   // UNICODE_TO_GBK[19826] := 16#71EC;
   // UNICODE_TO_GBK[19827] := 16#A053;
   // UNICODE_TO_GBK[19828] := 16#71ED;
   // UNICODE_TO_GBK[19829] := 16#A054;
   // UNICODE_TO_GBK[19830] := 16#71EE;
   // UNICODE_TO_GBK[19831] := 16#DBC6;
   // UNICODE_TO_GBK[19832] := 16#71EF;
   // UNICODE_TO_GBK[19833] := 16#A055;
   // UNICODE_TO_GBK[19834] := 16#71F0;
   // UNICODE_TO_GBK[19835] := 16#A056;
   // UNICODE_TO_GBK[19836] := 16#71F1;
   // UNICODE_TO_GBK[19837] := 16#A057;
   // UNICODE_TO_GBK[19838] := 16#71F2;
   // UNICODE_TO_GBK[19839] := 16#A058;
   // UNICODE_TO_GBK[19840] := 16#71F3;
   // UNICODE_TO_GBK[19841] := 16#A059;
   // UNICODE_TO_GBK[19842] := 16#71F4;
   // UNICODE_TO_GBK[19843] := 16#A05A;
   // UNICODE_TO_GBK[19844] := 16#71F5;
   // UNICODE_TO_GBK[19845] := 16#A05B;
   // UNICODE_TO_GBK[19846] := 16#71F6;
   // UNICODE_TO_GBK[19847] := 16#A05C;
   // UNICODE_TO_GBK[19848] := 16#71F7;
   // UNICODE_TO_GBK[19849] := 16#A05D;
   // UNICODE_TO_GBK[19850] := 16#71F8;
   // UNICODE_TO_GBK[19851] := 16#A05E;
   // UNICODE_TO_GBK[19852] := 16#71F9;
   // UNICODE_TO_GBK[19853] := 16#ECDE;
   // UNICODE_TO_GBK[19854] := 16#71FA;
   // UNICODE_TO_GBK[19855] := 16#A05F;
   // UNICODE_TO_GBK[19856] := 16#71FB;
   // UNICODE_TO_GBK[19857] := 16#A060;
   // UNICODE_TO_GBK[19858] := 16#71FC;
   // UNICODE_TO_GBK[19859] := 16#A061;
   // UNICODE_TO_GBK[19860] := 16#71FD;
   // UNICODE_TO_GBK[19861] := 16#A062;
   // UNICODE_TO_GBK[19862] := 16#71FE;
   // UNICODE_TO_GBK[19863] := 16#A063;
   // UNICODE_TO_GBK[19864] := 16#71FF;
   // UNICODE_TO_GBK[19865] := 16#A064;
   // UNICODE_TO_GBK[19866] := 16#7200;
   // UNICODE_TO_GBK[19867] := 16#A065;
   // UNICODE_TO_GBK[19868] := 16#7201;
   // UNICODE_TO_GBK[19869] := 16#A066;
   // UNICODE_TO_GBK[19870] := 16#7202;
   // UNICODE_TO_GBK[19871] := 16#A067;
   // UNICODE_TO_GBK[19872] := 16#7203;
   // UNICODE_TO_GBK[19873] := 16#A068;
   // UNICODE_TO_GBK[19874] := 16#7204;
   // UNICODE_TO_GBK[19875] := 16#A069;
   // UNICODE_TO_GBK[19876] := 16#7205;
   // UNICODE_TO_GBK[19877] := 16#A06A;
   // UNICODE_TO_GBK[19878] := 16#7206;
   // UNICODE_TO_GBK[19879] := 16#B1AC;
   // UNICODE_TO_GBK[19880] := 16#7207;
   // UNICODE_TO_GBK[19881] := 16#A06B;
   // UNICODE_TO_GBK[19882] := 16#7208;
   // UNICODE_TO_GBK[19883] := 16#A06C;
   // UNICODE_TO_GBK[19884] := 16#7209;
   // UNICODE_TO_GBK[19885] := 16#A06D;
   // UNICODE_TO_GBK[19886] := 16#720A;
   // UNICODE_TO_GBK[19887] := 16#A06E;
   // UNICODE_TO_GBK[19888] := 16#720B;
   // UNICODE_TO_GBK[19889] := 16#A06F;
   // UNICODE_TO_GBK[19890] := 16#720C;
   // UNICODE_TO_GBK[19891] := 16#A070;
   // UNICODE_TO_GBK[19892] := 16#720D;
   // UNICODE_TO_GBK[19893] := 16#A071;
   // UNICODE_TO_GBK[19894] := 16#720E;
   // UNICODE_TO_GBK[19895] := 16#A072;
   // UNICODE_TO_GBK[19896] := 16#720F;
   // UNICODE_TO_GBK[19897] := 16#A073;
   // UNICODE_TO_GBK[19898] := 16#7210;
   // UNICODE_TO_GBK[19899] := 16#A074;
   // UNICODE_TO_GBK[19900] := 16#7211;
   // UNICODE_TO_GBK[19901] := 16#A075;
   // UNICODE_TO_GBK[19902] := 16#7212;
   // UNICODE_TO_GBK[19903] := 16#A076;
   // UNICODE_TO_GBK[19904] := 16#7213;
   // UNICODE_TO_GBK[19905] := 16#A077;
   // UNICODE_TO_GBK[19906] := 16#7214;
   // UNICODE_TO_GBK[19907] := 16#A078;
   // UNICODE_TO_GBK[19908] := 16#7215;
   // UNICODE_TO_GBK[19909] := 16#A079;
   // UNICODE_TO_GBK[19910] := 16#7216;
   // UNICODE_TO_GBK[19911] := 16#A07A;
   // UNICODE_TO_GBK[19912] := 16#7217;
   // UNICODE_TO_GBK[19913] := 16#A07B;
   // UNICODE_TO_GBK[19914] := 16#7218;
   // UNICODE_TO_GBK[19915] := 16#A07C;
   // UNICODE_TO_GBK[19916] := 16#7219;
   // UNICODE_TO_GBK[19917] := 16#A07D;
   // UNICODE_TO_GBK[19918] := 16#721A;
   // UNICODE_TO_GBK[19919] := 16#A07E;
   // UNICODE_TO_GBK[19920] := 16#721B;
   // UNICODE_TO_GBK[19921] := 16#A080;
   // UNICODE_TO_GBK[19922] := 16#721C;
   // UNICODE_TO_GBK[19923] := 16#A081;
   // UNICODE_TO_GBK[19924] := 16#721D;
   // UNICODE_TO_GBK[19925] := 16#ECDF;
   // UNICODE_TO_GBK[19926] := 16#721E;
   // UNICODE_TO_GBK[19927] := 16#A082;
   // UNICODE_TO_GBK[19928] := 16#721F;
   // UNICODE_TO_GBK[19929] := 16#A083;
   // UNICODE_TO_GBK[19930] := 16#7220;
   // UNICODE_TO_GBK[19931] := 16#A084;
   // UNICODE_TO_GBK[19932] := 16#7221;
   // UNICODE_TO_GBK[19933] := 16#A085;
   // UNICODE_TO_GBK[19934] := 16#7222;
   // UNICODE_TO_GBK[19935] := 16#A086;
   // UNICODE_TO_GBK[19936] := 16#7223;
   // UNICODE_TO_GBK[19937] := 16#A087;
   // UNICODE_TO_GBK[19938] := 16#7224;
   // UNICODE_TO_GBK[19939] := 16#A088;
   // UNICODE_TO_GBK[19940] := 16#7225;
   // UNICODE_TO_GBK[19941] := 16#A089;
   // UNICODE_TO_GBK[19942] := 16#7226;
   // UNICODE_TO_GBK[19943] := 16#A08A;
   // UNICODE_TO_GBK[19944] := 16#7227;
   // UNICODE_TO_GBK[19945] := 16#A08B;
   // UNICODE_TO_GBK[19946] := 16#7228;
   // UNICODE_TO_GBK[19947] := 16#ECE0;
   // UNICODE_TO_GBK[19948] := 16#7229;
   // UNICODE_TO_GBK[19949] := 16#A08C;
   // UNICODE_TO_GBK[19950] := 16#722A;
   // UNICODE_TO_GBK[19951] := 16#D7A6;
   // UNICODE_TO_GBK[19952] := 16#722B;
   // UNICODE_TO_GBK[19953] := 16#A08D;
   // UNICODE_TO_GBK[19954] := 16#722C;
   // UNICODE_TO_GBK[19955] := 16#C5C0;
   // UNICODE_TO_GBK[19956] := 16#722D;
   // UNICODE_TO_GBK[19957] := 16#A08E;
   // UNICODE_TO_GBK[19958] := 16#722E;
   // UNICODE_TO_GBK[19959] := 16#A08F;
   // UNICODE_TO_GBK[19960] := 16#722F;
   // UNICODE_TO_GBK[19961] := 16#A090;
   // UNICODE_TO_GBK[19962] := 16#7230;
   // UNICODE_TO_GBK[19963] := 16#EBBC;
   // UNICODE_TO_GBK[19964] := 16#7231;
   // UNICODE_TO_GBK[19965] := 16#B0AE;
   // UNICODE_TO_GBK[19966] := 16#7232;
   // UNICODE_TO_GBK[19967] := 16#A091;
   // UNICODE_TO_GBK[19968] := 16#7233;
   // UNICODE_TO_GBK[19969] := 16#A092;
   // UNICODE_TO_GBK[19970] := 16#7234;
   // UNICODE_TO_GBK[19971] := 16#A093;
   // UNICODE_TO_GBK[19972] := 16#7235;
   // UNICODE_TO_GBK[19973] := 16#BEF4;
   // UNICODE_TO_GBK[19974] := 16#7236;
   // UNICODE_TO_GBK[19975] := 16#B8B8;
   // UNICODE_TO_GBK[19976] := 16#7237;
   // UNICODE_TO_GBK[19977] := 16#D2AF;
   // UNICODE_TO_GBK[19978] := 16#7238;
   // UNICODE_TO_GBK[19979] := 16#B0D6;
   // UNICODE_TO_GBK[19980] := 16#7239;
   // UNICODE_TO_GBK[19981] := 16#B5F9;
   // UNICODE_TO_GBK[19982] := 16#723A;
   // UNICODE_TO_GBK[19983] := 16#A094;
   // UNICODE_TO_GBK[19984] := 16#723B;
   // UNICODE_TO_GBK[19985] := 16#D8B3;
   // UNICODE_TO_GBK[19986] := 16#723C;
   // UNICODE_TO_GBK[19987] := 16#A095;
   // UNICODE_TO_GBK[19988] := 16#723D;
   // UNICODE_TO_GBK[19989] := 16#CBAC;
   // UNICODE_TO_GBK[19990] := 16#723E;
   // UNICODE_TO_GBK[19991] := 16#A096;
   // UNICODE_TO_GBK[19992] := 16#723F;
   // UNICODE_TO_GBK[19993] := 16#E3DD;
   // UNICODE_TO_GBK[19994] := 16#7240;
   // UNICODE_TO_GBK[19995] := 16#A097;
   // UNICODE_TO_GBK[19996] := 16#7241;
   // UNICODE_TO_GBK[19997] := 16#A098;
   // UNICODE_TO_GBK[19998] := 16#7242;
   // UNICODE_TO_GBK[19999] := 16#A099;
   // UNICODE_TO_GBK[20000] := 16#7243;
   // UNICODE_TO_GBK[20001] := 16#A09A;
   // UNICODE_TO_GBK[20002] := 16#7244;
   // UNICODE_TO_GBK[20003] := 16#A09B;
   // UNICODE_TO_GBK[20004] := 16#7245;
   // UNICODE_TO_GBK[20005] := 16#A09C;
   // UNICODE_TO_GBK[20006] := 16#7246;
   // UNICODE_TO_GBK[20007] := 16#A09D;
   // UNICODE_TO_GBK[20008] := 16#7247;
   // UNICODE_TO_GBK[20009] := 16#C6AC;
   // UNICODE_TO_GBK[20010] := 16#7248;
   // UNICODE_TO_GBK[20011] := 16#B0E6;
   // UNICODE_TO_GBK[20012] := 16#7249;
   // UNICODE_TO_GBK[20013] := 16#A09E;
   // UNICODE_TO_GBK[20014] := 16#724A;
   // UNICODE_TO_GBK[20015] := 16#A09F;
   // UNICODE_TO_GBK[20016] := 16#724B;
   // UNICODE_TO_GBK[20017] := 16#A0A0;
   // UNICODE_TO_GBK[20018] := 16#724C;
   // UNICODE_TO_GBK[20019] := 16#C5C6;
   // UNICODE_TO_GBK[20020] := 16#724D;
   // UNICODE_TO_GBK[20021] := 16#EBB9;
   // UNICODE_TO_GBK[20022] := 16#724E;
   // UNICODE_TO_GBK[20023] := 16#A0A1;
   // UNICODE_TO_GBK[20024] := 16#724F;
   // UNICODE_TO_GBK[20025] := 16#A0A2;
   // UNICODE_TO_GBK[20026] := 16#7250;
   // UNICODE_TO_GBK[20027] := 16#A0A3;
   // UNICODE_TO_GBK[20028] := 16#7251;
   // UNICODE_TO_GBK[20029] := 16#A0A4;
   // UNICODE_TO_GBK[20030] := 16#7252;
   // UNICODE_TO_GBK[20031] := 16#EBBA;
   // UNICODE_TO_GBK[20032] := 16#7253;
   // UNICODE_TO_GBK[20033] := 16#A0A5;
   // UNICODE_TO_GBK[20034] := 16#7254;
   // UNICODE_TO_GBK[20035] := 16#A0A6;
   // UNICODE_TO_GBK[20036] := 16#7255;
   // UNICODE_TO_GBK[20037] := 16#A0A7;
   // UNICODE_TO_GBK[20038] := 16#7256;
   // UNICODE_TO_GBK[20039] := 16#EBBB;
   // UNICODE_TO_GBK[20040] := 16#7257;
   // UNICODE_TO_GBK[20041] := 16#A0A8;
   // UNICODE_TO_GBK[20042] := 16#7258;
   // UNICODE_TO_GBK[20043] := 16#A0A9;
   // UNICODE_TO_GBK[20044] := 16#7259;
   // UNICODE_TO_GBK[20045] := 16#D1C0;
   // UNICODE_TO_GBK[20046] := 16#725A;
   // UNICODE_TO_GBK[20047] := 16#A0AA;
   // UNICODE_TO_GBK[20048] := 16#725B;
   // UNICODE_TO_GBK[20049] := 16#C5A3;
   // UNICODE_TO_GBK[20050] := 16#725C;
   // UNICODE_TO_GBK[20051] := 16#A0AB;
   // UNICODE_TO_GBK[20052] := 16#725D;
   // UNICODE_TO_GBK[20053] := 16#EAF2;
   // UNICODE_TO_GBK[20054] := 16#725E;
   // UNICODE_TO_GBK[20055] := 16#A0AC;
   // UNICODE_TO_GBK[20056] := 16#725F;
   // UNICODE_TO_GBK[20057] := 16#C4B2;
   // UNICODE_TO_GBK[20058] := 16#7260;
   // UNICODE_TO_GBK[20059] := 16#A0AD;
   // UNICODE_TO_GBK[20060] := 16#7261;
   // UNICODE_TO_GBK[20061] := 16#C4B5;
   // UNICODE_TO_GBK[20062] := 16#7262;
   // UNICODE_TO_GBK[20063] := 16#C0CE;
   // UNICODE_TO_GBK[20064] := 16#7263;
   // UNICODE_TO_GBK[20065] := 16#A0AE;
   // UNICODE_TO_GBK[20066] := 16#7264;
   // UNICODE_TO_GBK[20067] := 16#A0AF;
   // UNICODE_TO_GBK[20068] := 16#7265;
   // UNICODE_TO_GBK[20069] := 16#A0B0;
   // UNICODE_TO_GBK[20070] := 16#7266;
   // UNICODE_TO_GBK[20071] := 16#EAF3;
   // UNICODE_TO_GBK[20072] := 16#7267;
   // UNICODE_TO_GBK[20073] := 16#C4C1;
   // UNICODE_TO_GBK[20074] := 16#7268;
   // UNICODE_TO_GBK[20075] := 16#A0B1;
   // UNICODE_TO_GBK[20076] := 16#7269;
   // UNICODE_TO_GBK[20077] := 16#CEEF;
   // UNICODE_TO_GBK[20078] := 16#726A;
   // UNICODE_TO_GBK[20079] := 16#A0B2;
   // UNICODE_TO_GBK[20080] := 16#726B;
   // UNICODE_TO_GBK[20081] := 16#A0B3;
   // UNICODE_TO_GBK[20082] := 16#726C;
   // UNICODE_TO_GBK[20083] := 16#A0B4;
   // UNICODE_TO_GBK[20084] := 16#726D;
   // UNICODE_TO_GBK[20085] := 16#A0B5;
   // UNICODE_TO_GBK[20086] := 16#726E;
   // UNICODE_TO_GBK[20087] := 16#EAF0;
   // UNICODE_TO_GBK[20088] := 16#726F;
   // UNICODE_TO_GBK[20089] := 16#EAF4;
   // UNICODE_TO_GBK[20090] := 16#7270;
   // UNICODE_TO_GBK[20091] := 16#A0B6;
   // UNICODE_TO_GBK[20092] := 16#7271;
   // UNICODE_TO_GBK[20093] := 16#A0B7;
   // UNICODE_TO_GBK[20094] := 16#7272;
   // UNICODE_TO_GBK[20095] := 16#C9FC;
   // UNICODE_TO_GBK[20096] := 16#7273;
   // UNICODE_TO_GBK[20097] := 16#A0B8;
   // UNICODE_TO_GBK[20098] := 16#7274;
   // UNICODE_TO_GBK[20099] := 16#A0B9;
   // UNICODE_TO_GBK[20100] := 16#7275;
   // UNICODE_TO_GBK[20101] := 16#C7A3;
   // UNICODE_TO_GBK[20102] := 16#7276;
   // UNICODE_TO_GBK[20103] := 16#A0BA;
   // UNICODE_TO_GBK[20104] := 16#7277;
   // UNICODE_TO_GBK[20105] := 16#A0BB;
   // UNICODE_TO_GBK[20106] := 16#7278;
   // UNICODE_TO_GBK[20107] := 16#A0BC;
   // UNICODE_TO_GBK[20108] := 16#7279;
   // UNICODE_TO_GBK[20109] := 16#CCD8;
   // UNICODE_TO_GBK[20110] := 16#727A;
   // UNICODE_TO_GBK[20111] := 16#CEFE;
   // UNICODE_TO_GBK[20112] := 16#727B;
   // UNICODE_TO_GBK[20113] := 16#A0BD;
   // UNICODE_TO_GBK[20114] := 16#727C;
   // UNICODE_TO_GBK[20115] := 16#A0BE;
   // UNICODE_TO_GBK[20116] := 16#727D;
   // UNICODE_TO_GBK[20117] := 16#A0BF;
   // UNICODE_TO_GBK[20118] := 16#727E;
   // UNICODE_TO_GBK[20119] := 16#EAF5;
   // UNICODE_TO_GBK[20120] := 16#727F;
   // UNICODE_TO_GBK[20121] := 16#EAF6;
   // UNICODE_TO_GBK[20122] := 16#7280;
   // UNICODE_TO_GBK[20123] := 16#CFAC;
   // UNICODE_TO_GBK[20124] := 16#7281;
   // UNICODE_TO_GBK[20125] := 16#C0E7;
   // UNICODE_TO_GBK[20126] := 16#7282;
   // UNICODE_TO_GBK[20127] := 16#A0C0;
   // UNICODE_TO_GBK[20128] := 16#7283;
   // UNICODE_TO_GBK[20129] := 16#A0C1;
   // UNICODE_TO_GBK[20130] := 16#7284;
   // UNICODE_TO_GBK[20131] := 16#EAF7;
   // UNICODE_TO_GBK[20132] := 16#7285;
   // UNICODE_TO_GBK[20133] := 16#A0C2;
   // UNICODE_TO_GBK[20134] := 16#7286;
   // UNICODE_TO_GBK[20135] := 16#A0C3;
   // UNICODE_TO_GBK[20136] := 16#7287;
   // UNICODE_TO_GBK[20137] := 16#A0C4;
   // UNICODE_TO_GBK[20138] := 16#7288;
   // UNICODE_TO_GBK[20139] := 16#A0C5;
   // UNICODE_TO_GBK[20140] := 16#7289;
   // UNICODE_TO_GBK[20141] := 16#A0C6;
   // UNICODE_TO_GBK[20142] := 16#728A;
   // UNICODE_TO_GBK[20143] := 16#B6BF;
   // UNICODE_TO_GBK[20144] := 16#728B;
   // UNICODE_TO_GBK[20145] := 16#EAF8;
   // UNICODE_TO_GBK[20146] := 16#728C;
   // UNICODE_TO_GBK[20147] := 16#A0C7;
   // UNICODE_TO_GBK[20148] := 16#728D;
   // UNICODE_TO_GBK[20149] := 16#EAF9;
   // UNICODE_TO_GBK[20150] := 16#728E;
   // UNICODE_TO_GBK[20151] := 16#A0C8;
   // UNICODE_TO_GBK[20152] := 16#728F;
   // UNICODE_TO_GBK[20153] := 16#EAFA;
   // UNICODE_TO_GBK[20154] := 16#7290;
   // UNICODE_TO_GBK[20155] := 16#A0C9;
   // UNICODE_TO_GBK[20156] := 16#7291;
   // UNICODE_TO_GBK[20157] := 16#A0CA;
   // UNICODE_TO_GBK[20158] := 16#7292;
   // UNICODE_TO_GBK[20159] := 16#EAFB;
   // UNICODE_TO_GBK[20160] := 16#7293;
   // UNICODE_TO_GBK[20161] := 16#A0CB;
   // UNICODE_TO_GBK[20162] := 16#7294;
   // UNICODE_TO_GBK[20163] := 16#A0CC;
   // UNICODE_TO_GBK[20164] := 16#7295;
   // UNICODE_TO_GBK[20165] := 16#A0CD;
   // UNICODE_TO_GBK[20166] := 16#7296;
   // UNICODE_TO_GBK[20167] := 16#A0CE;
   // UNICODE_TO_GBK[20168] := 16#7297;
   // UNICODE_TO_GBK[20169] := 16#A0CF;
   // UNICODE_TO_GBK[20170] := 16#7298;
   // UNICODE_TO_GBK[20171] := 16#A0D0;
   // UNICODE_TO_GBK[20172] := 16#7299;
   // UNICODE_TO_GBK[20173] := 16#A0D1;
   // UNICODE_TO_GBK[20174] := 16#729A;
   // UNICODE_TO_GBK[20175] := 16#A0D2;
   // UNICODE_TO_GBK[20176] := 16#729B;
   // UNICODE_TO_GBK[20177] := 16#A0D3;
   // UNICODE_TO_GBK[20178] := 16#729C;
   // UNICODE_TO_GBK[20179] := 16#A0D4;
   // UNICODE_TO_GBK[20180] := 16#729D;
   // UNICODE_TO_GBK[20181] := 16#A0D5;
   // UNICODE_TO_GBK[20182] := 16#729E;
   // UNICODE_TO_GBK[20183] := 16#A0D6;
   // UNICODE_TO_GBK[20184] := 16#729F;
   // UNICODE_TO_GBK[20185] := 16#EAF1;
   // UNICODE_TO_GBK[20186] := 16#72A0;
   // UNICODE_TO_GBK[20187] := 16#A0D7;
   // UNICODE_TO_GBK[20188] := 16#72A1;
   // UNICODE_TO_GBK[20189] := 16#A0D8;
   // UNICODE_TO_GBK[20190] := 16#72A2;
   // UNICODE_TO_GBK[20191] := 16#A0D9;
   // UNICODE_TO_GBK[20192] := 16#72A3;
   // UNICODE_TO_GBK[20193] := 16#A0DA;
   // UNICODE_TO_GBK[20194] := 16#72A4;
   // UNICODE_TO_GBK[20195] := 16#A0DB;
   // UNICODE_TO_GBK[20196] := 16#72A5;
   // UNICODE_TO_GBK[20197] := 16#A0DC;
   // UNICODE_TO_GBK[20198] := 16#72A6;
   // UNICODE_TO_GBK[20199] := 16#A0DD;
   // UNICODE_TO_GBK[20200] := 16#72A7;
   // UNICODE_TO_GBK[20201] := 16#A0DE;
   // UNICODE_TO_GBK[20202] := 16#72A8;
   // UNICODE_TO_GBK[20203] := 16#A0DF;
   // UNICODE_TO_GBK[20204] := 16#72A9;
   // UNICODE_TO_GBK[20205] := 16#A0E0;
   // UNICODE_TO_GBK[20206] := 16#72AA;
   // UNICODE_TO_GBK[20207] := 16#A0E1;
   // UNICODE_TO_GBK[20208] := 16#72AB;
   // UNICODE_TO_GBK[20209] := 16#A0E2;
   // UNICODE_TO_GBK[20210] := 16#72AC;
   // UNICODE_TO_GBK[20211] := 16#C8AE;
   // UNICODE_TO_GBK[20212] := 16#72AD;
   // UNICODE_TO_GBK[20213] := 16#E1EB;
   // UNICODE_TO_GBK[20214] := 16#72AE;
   // UNICODE_TO_GBK[20215] := 16#A0E3;
   // UNICODE_TO_GBK[20216] := 16#72AF;
   // UNICODE_TO_GBK[20217] := 16#B7B8;
   // UNICODE_TO_GBK[20218] := 16#72B0;
   // UNICODE_TO_GBK[20219] := 16#E1EC;
   // UNICODE_TO_GBK[20220] := 16#72B1;
   // UNICODE_TO_GBK[20221] := 16#A0E4;
   // UNICODE_TO_GBK[20222] := 16#72B2;
   // UNICODE_TO_GBK[20223] := 16#A0E5;
   // UNICODE_TO_GBK[20224] := 16#72B3;
   // UNICODE_TO_GBK[20225] := 16#A0E6;
   // UNICODE_TO_GBK[20226] := 16#72B4;
   // UNICODE_TO_GBK[20227] := 16#E1ED;
   // UNICODE_TO_GBK[20228] := 16#72B5;
   // UNICODE_TO_GBK[20229] := 16#A0E7;
   // UNICODE_TO_GBK[20230] := 16#72B6;
   // UNICODE_TO_GBK[20231] := 16#D7B4;
   // UNICODE_TO_GBK[20232] := 16#72B7;
   // UNICODE_TO_GBK[20233] := 16#E1EE;
   // UNICODE_TO_GBK[20234] := 16#72B8;
   // UNICODE_TO_GBK[20235] := 16#E1EF;
   // UNICODE_TO_GBK[20236] := 16#72B9;
   // UNICODE_TO_GBK[20237] := 16#D3CC;
   // UNICODE_TO_GBK[20238] := 16#72BA;
   // UNICODE_TO_GBK[20239] := 16#A0E8;
   // UNICODE_TO_GBK[20240] := 16#72BB;
   // UNICODE_TO_GBK[20241] := 16#A0E9;
   // UNICODE_TO_GBK[20242] := 16#72BC;
   // UNICODE_TO_GBK[20243] := 16#A0EA;
   // UNICODE_TO_GBK[20244] := 16#72BD;
   // UNICODE_TO_GBK[20245] := 16#A0EB;
   // UNICODE_TO_GBK[20246] := 16#72BE;
   // UNICODE_TO_GBK[20247] := 16#A0EC;
   // UNICODE_TO_GBK[20248] := 16#72BF;
   // UNICODE_TO_GBK[20249] := 16#A0ED;
   // UNICODE_TO_GBK[20250] := 16#72C0;
   // UNICODE_TO_GBK[20251] := 16#A0EE;
   // UNICODE_TO_GBK[20252] := 16#72C1;
   // UNICODE_TO_GBK[20253] := 16#E1F1;
   // UNICODE_TO_GBK[20254] := 16#72C2;
   // UNICODE_TO_GBK[20255] := 16#BFF1;
   // UNICODE_TO_GBK[20256] := 16#72C3;
   // UNICODE_TO_GBK[20257] := 16#E1F0;
   // UNICODE_TO_GBK[20258] := 16#72C4;
   // UNICODE_TO_GBK[20259] := 16#B5D2;
   // UNICODE_TO_GBK[20260] := 16#72C5;
   // UNICODE_TO_GBK[20261] := 16#A0EF;
   // UNICODE_TO_GBK[20262] := 16#72C6;
   // UNICODE_TO_GBK[20263] := 16#A0F0;
   // UNICODE_TO_GBK[20264] := 16#72C7;
   // UNICODE_TO_GBK[20265] := 16#A0F1;
   // UNICODE_TO_GBK[20266] := 16#72C8;
   // UNICODE_TO_GBK[20267] := 16#B1B7;
   // UNICODE_TO_GBK[20268] := 16#72C9;
   // UNICODE_TO_GBK[20269] := 16#A0F2;
   // UNICODE_TO_GBK[20270] := 16#72CA;
   // UNICODE_TO_GBK[20271] := 16#A0F3;
   // UNICODE_TO_GBK[20272] := 16#72CB;
   // UNICODE_TO_GBK[20273] := 16#A0F4;
   // UNICODE_TO_GBK[20274] := 16#72CC;
   // UNICODE_TO_GBK[20275] := 16#A0F5;
   // UNICODE_TO_GBK[20276] := 16#72CD;
   // UNICODE_TO_GBK[20277] := 16#E1F3;
   // UNICODE_TO_GBK[20278] := 16#72CE;
   // UNICODE_TO_GBK[20279] := 16#E1F2;
   // UNICODE_TO_GBK[20280] := 16#72CF;
   // UNICODE_TO_GBK[20281] := 16#A0F6;
   // UNICODE_TO_GBK[20282] := 16#72D0;
   // UNICODE_TO_GBK[20283] := 16#BAFC;
   // UNICODE_TO_GBK[20284] := 16#72D1;
   // UNICODE_TO_GBK[20285] := 16#A0F7;
   // UNICODE_TO_GBK[20286] := 16#72D2;
   // UNICODE_TO_GBK[20287] := 16#E1F4;
   // UNICODE_TO_GBK[20288] := 16#72D3;
   // UNICODE_TO_GBK[20289] := 16#A0F8;
   // UNICODE_TO_GBK[20290] := 16#72D4;
   // UNICODE_TO_GBK[20291] := 16#A0F9;
   // UNICODE_TO_GBK[20292] := 16#72D5;
   // UNICODE_TO_GBK[20293] := 16#A0FA;
   // UNICODE_TO_GBK[20294] := 16#72D6;
   // UNICODE_TO_GBK[20295] := 16#A0FB;
   // UNICODE_TO_GBK[20296] := 16#72D7;
   // UNICODE_TO_GBK[20297] := 16#B9B7;
   // UNICODE_TO_GBK[20298] := 16#72D8;
   // UNICODE_TO_GBK[20299] := 16#A0FC;
   // UNICODE_TO_GBK[20300] := 16#72D9;
   // UNICODE_TO_GBK[20301] := 16#BED1;
   // UNICODE_TO_GBK[20302] := 16#72DA;
   // UNICODE_TO_GBK[20303] := 16#A0FD;
   // UNICODE_TO_GBK[20304] := 16#72DB;
   // UNICODE_TO_GBK[20305] := 16#A0FE;
   // UNICODE_TO_GBK[20306] := 16#72DC;
   // UNICODE_TO_GBK[20307] := 16#AA40;
   // UNICODE_TO_GBK[20308] := 16#72DD;
   // UNICODE_TO_GBK[20309] := 16#AA41;
   // UNICODE_TO_GBK[20310] := 16#72DE;
   // UNICODE_TO_GBK[20311] := 16#C4FC;
   // UNICODE_TO_GBK[20312] := 16#72DF;
   // UNICODE_TO_GBK[20313] := 16#AA42;
   // UNICODE_TO_GBK[20314] := 16#72E0;
   // UNICODE_TO_GBK[20315] := 16#BADD;
   // UNICODE_TO_GBK[20316] := 16#72E1;
   // UNICODE_TO_GBK[20317] := 16#BDC6;
   // UNICODE_TO_GBK[20318] := 16#72E2;
   // UNICODE_TO_GBK[20319] := 16#AA43;
   // UNICODE_TO_GBK[20320] := 16#72E3;
   // UNICODE_TO_GBK[20321] := 16#AA44;
   // UNICODE_TO_GBK[20322] := 16#72E4;
   // UNICODE_TO_GBK[20323] := 16#AA45;
   // UNICODE_TO_GBK[20324] := 16#72E5;
   // UNICODE_TO_GBK[20325] := 16#AA46;
   // UNICODE_TO_GBK[20326] := 16#72E6;
   // UNICODE_TO_GBK[20327] := 16#AA47;
   // UNICODE_TO_GBK[20328] := 16#72E7;
   // UNICODE_TO_GBK[20329] := 16#AA48;
   // UNICODE_TO_GBK[20330] := 16#72E8;
   // UNICODE_TO_GBK[20331] := 16#E1F5;
   // UNICODE_TO_GBK[20332] := 16#72E9;
   // UNICODE_TO_GBK[20333] := 16#E1F7;
   // UNICODE_TO_GBK[20334] := 16#72EA;
   // UNICODE_TO_GBK[20335] := 16#AA49;
   // UNICODE_TO_GBK[20336] := 16#72EB;
   // UNICODE_TO_GBK[20337] := 16#AA4A;
   // UNICODE_TO_GBK[20338] := 16#72EC;
   // UNICODE_TO_GBK[20339] := 16#B6C0;
   // UNICODE_TO_GBK[20340] := 16#72ED;
   // UNICODE_TO_GBK[20341] := 16#CFC1;
   // UNICODE_TO_GBK[20342] := 16#72EE;
   // UNICODE_TO_GBK[20343] := 16#CAA8;
   // UNICODE_TO_GBK[20344] := 16#72EF;
   // UNICODE_TO_GBK[20345] := 16#E1F6;
   // UNICODE_TO_GBK[20346] := 16#72F0;
   // UNICODE_TO_GBK[20347] := 16#D5F8;
   // UNICODE_TO_GBK[20348] := 16#72F1;
   // UNICODE_TO_GBK[20349] := 16#D3FC;
   // UNICODE_TO_GBK[20350] := 16#72F2;
   // UNICODE_TO_GBK[20351] := 16#E1F8;
   // UNICODE_TO_GBK[20352] := 16#72F3;
   // UNICODE_TO_GBK[20353] := 16#E1FC;
   // UNICODE_TO_GBK[20354] := 16#72F4;
   // UNICODE_TO_GBK[20355] := 16#E1F9;
   // UNICODE_TO_GBK[20356] := 16#72F5;
   // UNICODE_TO_GBK[20357] := 16#AA4B;
   // UNICODE_TO_GBK[20358] := 16#72F6;
   // UNICODE_TO_GBK[20359] := 16#AA4C;
   // UNICODE_TO_GBK[20360] := 16#72F7;
   // UNICODE_TO_GBK[20361] := 16#E1FA;
   // UNICODE_TO_GBK[20362] := 16#72F8;
   // UNICODE_TO_GBK[20363] := 16#C0EA;
   // UNICODE_TO_GBK[20364] := 16#72F9;
   // UNICODE_TO_GBK[20365] := 16#AA4D;
   // UNICODE_TO_GBK[20366] := 16#72FA;
   // UNICODE_TO_GBK[20367] := 16#E1FE;
   // UNICODE_TO_GBK[20368] := 16#72FB;
   // UNICODE_TO_GBK[20369] := 16#E2A1;
   // UNICODE_TO_GBK[20370] := 16#72FC;
   // UNICODE_TO_GBK[20371] := 16#C0C7;
   // UNICODE_TO_GBK[20372] := 16#72FD;
   // UNICODE_TO_GBK[20373] := 16#AA4E;
   // UNICODE_TO_GBK[20374] := 16#72FE;
   // UNICODE_TO_GBK[20375] := 16#AA4F;
   // UNICODE_TO_GBK[20376] := 16#72FF;
   // UNICODE_TO_GBK[20377] := 16#AA50;
   // UNICODE_TO_GBK[20378] := 16#7300;
   // UNICODE_TO_GBK[20379] := 16#AA51;
   // UNICODE_TO_GBK[20380] := 16#7301;
   // UNICODE_TO_GBK[20381] := 16#E1FB;
   // UNICODE_TO_GBK[20382] := 16#7302;
   // UNICODE_TO_GBK[20383] := 16#AA52;
   // UNICODE_TO_GBK[20384] := 16#7303;
   // UNICODE_TO_GBK[20385] := 16#E1FD;
   // UNICODE_TO_GBK[20386] := 16#7304;
   // UNICODE_TO_GBK[20387] := 16#AA53;
   // UNICODE_TO_GBK[20388] := 16#7305;
   // UNICODE_TO_GBK[20389] := 16#AA54;
   // UNICODE_TO_GBK[20390] := 16#7306;
   // UNICODE_TO_GBK[20391] := 16#AA55;
   // UNICODE_TO_GBK[20392] := 16#7307;
   // UNICODE_TO_GBK[20393] := 16#AA56;
   // UNICODE_TO_GBK[20394] := 16#7308;
   // UNICODE_TO_GBK[20395] := 16#AA57;
   // UNICODE_TO_GBK[20396] := 16#7309;
   // UNICODE_TO_GBK[20397] := 16#AA58;
   // UNICODE_TO_GBK[20398] := 16#730A;
   // UNICODE_TO_GBK[20399] := 16#E2A5;
   // UNICODE_TO_GBK[20400] := 16#730B;
   // UNICODE_TO_GBK[20401] := 16#AA59;
   // UNICODE_TO_GBK[20402] := 16#730C;
   // UNICODE_TO_GBK[20403] := 16#AA5A;
   // UNICODE_TO_GBK[20404] := 16#730D;
   // UNICODE_TO_GBK[20405] := 16#AA5B;
   // UNICODE_TO_GBK[20406] := 16#730E;
   // UNICODE_TO_GBK[20407] := 16#C1D4;
   // UNICODE_TO_GBK[20408] := 16#730F;
   // UNICODE_TO_GBK[20409] := 16#AA5C;
   // UNICODE_TO_GBK[20410] := 16#7310;
   // UNICODE_TO_GBK[20411] := 16#AA5D;
   // UNICODE_TO_GBK[20412] := 16#7311;
   // UNICODE_TO_GBK[20413] := 16#AA5E;
   // UNICODE_TO_GBK[20414] := 16#7312;
   // UNICODE_TO_GBK[20415] := 16#AA5F;
   // UNICODE_TO_GBK[20416] := 16#7313;
   // UNICODE_TO_GBK[20417] := 16#E2A3;
   // UNICODE_TO_GBK[20418] := 16#7314;
   // UNICODE_TO_GBK[20419] := 16#AA60;
   // UNICODE_TO_GBK[20420] := 16#7315;
   // UNICODE_TO_GBK[20421] := 16#E2A8;
   // UNICODE_TO_GBK[20422] := 16#7316;
   // UNICODE_TO_GBK[20423] := 16#B2FE;
   // UNICODE_TO_GBK[20424] := 16#7317;
   // UNICODE_TO_GBK[20425] := 16#E2A2;
   // UNICODE_TO_GBK[20426] := 16#7318;
   // UNICODE_TO_GBK[20427] := 16#AA61;
   // UNICODE_TO_GBK[20428] := 16#7319;
   // UNICODE_TO_GBK[20429] := 16#AA62;
   // UNICODE_TO_GBK[20430] := 16#731A;
   // UNICODE_TO_GBK[20431] := 16#AA63;
   // UNICODE_TO_GBK[20432] := 16#731B;
   // UNICODE_TO_GBK[20433] := 16#C3CD;
   // UNICODE_TO_GBK[20434] := 16#731C;
   // UNICODE_TO_GBK[20435] := 16#B2C2;
   // UNICODE_TO_GBK[20436] := 16#731D;
   // UNICODE_TO_GBK[20437] := 16#E2A7;
   // UNICODE_TO_GBK[20438] := 16#731E;
   // UNICODE_TO_GBK[20439] := 16#E2A6;
   // UNICODE_TO_GBK[20440] := 16#731F;
   // UNICODE_TO_GBK[20441] := 16#AA64;
   // UNICODE_TO_GBK[20442] := 16#7320;
   // UNICODE_TO_GBK[20443] := 16#AA65;
   // UNICODE_TO_GBK[20444] := 16#7321;
   // UNICODE_TO_GBK[20445] := 16#E2A4;
   // UNICODE_TO_GBK[20446] := 16#7322;
   // UNICODE_TO_GBK[20447] := 16#E2A9;
   // UNICODE_TO_GBK[20448] := 16#7323;
   // UNICODE_TO_GBK[20449] := 16#AA66;
   // UNICODE_TO_GBK[20450] := 16#7324;
   // UNICODE_TO_GBK[20451] := 16#AA67;
   // UNICODE_TO_GBK[20452] := 16#7325;
   // UNICODE_TO_GBK[20453] := 16#E2AB;
   // UNICODE_TO_GBK[20454] := 16#7326;
   // UNICODE_TO_GBK[20455] := 16#AA68;
   // UNICODE_TO_GBK[20456] := 16#7327;
   // UNICODE_TO_GBK[20457] := 16#AA69;
   // UNICODE_TO_GBK[20458] := 16#7328;
   // UNICODE_TO_GBK[20459] := 16#AA6A;
   // UNICODE_TO_GBK[20460] := 16#7329;
   // UNICODE_TO_GBK[20461] := 16#D0C9;
   // UNICODE_TO_GBK[20462] := 16#732A;
   // UNICODE_TO_GBK[20463] := 16#D6ED;
   // UNICODE_TO_GBK[20464] := 16#732B;
   // UNICODE_TO_GBK[20465] := 16#C3A8;
   // UNICODE_TO_GBK[20466] := 16#732C;
   // UNICODE_TO_GBK[20467] := 16#E2AC;
   // UNICODE_TO_GBK[20468] := 16#732D;
   // UNICODE_TO_GBK[20469] := 16#AA6B;
   // UNICODE_TO_GBK[20470] := 16#732E;
   // UNICODE_TO_GBK[20471] := 16#CFD7;
   // UNICODE_TO_GBK[20472] := 16#732F;
   // UNICODE_TO_GBK[20473] := 16#AA6C;
   // UNICODE_TO_GBK[20474] := 16#7330;
   // UNICODE_TO_GBK[20475] := 16#AA6D;
   // UNICODE_TO_GBK[20476] := 16#7331;
   // UNICODE_TO_GBK[20477] := 16#E2AE;
   // UNICODE_TO_GBK[20478] := 16#7332;
   // UNICODE_TO_GBK[20479] := 16#AA6E;
   // UNICODE_TO_GBK[20480] := 16#7333;
   // UNICODE_TO_GBK[20481] := 16#AA6F;
   // UNICODE_TO_GBK[20482] := 16#7334;
   // UNICODE_TO_GBK[20483] := 16#BAEF;
   // UNICODE_TO_GBK[20484] := 16#7335;
   // UNICODE_TO_GBK[20485] := 16#AA70;
   // UNICODE_TO_GBK[20486] := 16#7336;
   // UNICODE_TO_GBK[20487] := 16#AA71;
   // UNICODE_TO_GBK[20488] := 16#7337;
   // UNICODE_TO_GBK[20489] := 16#E9E0;
   // UNICODE_TO_GBK[20490] := 16#7338;
   // UNICODE_TO_GBK[20491] := 16#E2AD;
   // UNICODE_TO_GBK[20492] := 16#7339;
   // UNICODE_TO_GBK[20493] := 16#E2AA;
   // UNICODE_TO_GBK[20494] := 16#733A;
   // UNICODE_TO_GBK[20495] := 16#AA72;
   // UNICODE_TO_GBK[20496] := 16#733B;
   // UNICODE_TO_GBK[20497] := 16#AA73;
   // UNICODE_TO_GBK[20498] := 16#733C;
   // UNICODE_TO_GBK[20499] := 16#AA74;
   // UNICODE_TO_GBK[20500] := 16#733D;
   // UNICODE_TO_GBK[20501] := 16#AA75;
   // UNICODE_TO_GBK[20502] := 16#733E;
   // UNICODE_TO_GBK[20503] := 16#BBAB;
   // UNICODE_TO_GBK[20504] := 16#733F;
   // UNICODE_TO_GBK[20505] := 16#D4B3;
   // UNICODE_TO_GBK[20506] := 16#7340;
   // UNICODE_TO_GBK[20507] := 16#AA76;
   // UNICODE_TO_GBK[20508] := 16#7341;
   // UNICODE_TO_GBK[20509] := 16#AA77;
   // UNICODE_TO_GBK[20510] := 16#7342;
   // UNICODE_TO_GBK[20511] := 16#AA78;
   // UNICODE_TO_GBK[20512] := 16#7343;
   // UNICODE_TO_GBK[20513] := 16#AA79;
   // UNICODE_TO_GBK[20514] := 16#7344;
   // UNICODE_TO_GBK[20515] := 16#AA7A;
   // UNICODE_TO_GBK[20516] := 16#7345;
   // UNICODE_TO_GBK[20517] := 16#AA7B;
   // UNICODE_TO_GBK[20518] := 16#7346;
   // UNICODE_TO_GBK[20519] := 16#AA7C;
   // UNICODE_TO_GBK[20520] := 16#7347;
   // UNICODE_TO_GBK[20521] := 16#AA7D;
   // UNICODE_TO_GBK[20522] := 16#7348;
   // UNICODE_TO_GBK[20523] := 16#AA7E;
   // UNICODE_TO_GBK[20524] := 16#7349;
   // UNICODE_TO_GBK[20525] := 16#AA80;
   // UNICODE_TO_GBK[20526] := 16#734A;
   // UNICODE_TO_GBK[20527] := 16#AA81;
   // UNICODE_TO_GBK[20528] := 16#734B;
   // UNICODE_TO_GBK[20529] := 16#AA82;
   // UNICODE_TO_GBK[20530] := 16#734C;
   // UNICODE_TO_GBK[20531] := 16#AA83;
   // UNICODE_TO_GBK[20532] := 16#734D;
   // UNICODE_TO_GBK[20533] := 16#E2B0;
   // UNICODE_TO_GBK[20534] := 16#734E;
   // UNICODE_TO_GBK[20535] := 16#AA84;
   // UNICODE_TO_GBK[20536] := 16#734F;
   // UNICODE_TO_GBK[20537] := 16#AA85;
   // UNICODE_TO_GBK[20538] := 16#7350;
   // UNICODE_TO_GBK[20539] := 16#E2AF;
   // UNICODE_TO_GBK[20540] := 16#7351;
   // UNICODE_TO_GBK[20541] := 16#AA86;
   // UNICODE_TO_GBK[20542] := 16#7352;
   // UNICODE_TO_GBK[20543] := 16#E9E1;
   // UNICODE_TO_GBK[20544] := 16#7353;
   // UNICODE_TO_GBK[20545] := 16#AA87;
   // UNICODE_TO_GBK[20546] := 16#7354;
   // UNICODE_TO_GBK[20547] := 16#AA88;
   // UNICODE_TO_GBK[20548] := 16#7355;
   // UNICODE_TO_GBK[20549] := 16#AA89;
   // UNICODE_TO_GBK[20550] := 16#7356;
   // UNICODE_TO_GBK[20551] := 16#AA8A;
   // UNICODE_TO_GBK[20552] := 16#7357;
   // UNICODE_TO_GBK[20553] := 16#E2B1;
   // UNICODE_TO_GBK[20554] := 16#7358;
   // UNICODE_TO_GBK[20555] := 16#AA8B;
   // UNICODE_TO_GBK[20556] := 16#7359;
   // UNICODE_TO_GBK[20557] := 16#AA8C;
   // UNICODE_TO_GBK[20558] := 16#735A;
   // UNICODE_TO_GBK[20559] := 16#AA8D;
   // UNICODE_TO_GBK[20560] := 16#735B;
   // UNICODE_TO_GBK[20561] := 16#AA8E;
   // UNICODE_TO_GBK[20562] := 16#735C;
   // UNICODE_TO_GBK[20563] := 16#AA8F;
   // UNICODE_TO_GBK[20564] := 16#735D;
   // UNICODE_TO_GBK[20565] := 16#AA90;
   // UNICODE_TO_GBK[20566] := 16#735E;
   // UNICODE_TO_GBK[20567] := 16#AA91;
   // UNICODE_TO_GBK[20568] := 16#735F;
   // UNICODE_TO_GBK[20569] := 16#AA92;
   // UNICODE_TO_GBK[20570] := 16#7360;
   // UNICODE_TO_GBK[20571] := 16#E2B2;
   // UNICODE_TO_GBK[20572] := 16#7361;
   // UNICODE_TO_GBK[20573] := 16#AA93;
   // UNICODE_TO_GBK[20574] := 16#7362;
   // UNICODE_TO_GBK[20575] := 16#AA94;
   // UNICODE_TO_GBK[20576] := 16#7363;
   // UNICODE_TO_GBK[20577] := 16#AA95;
   // UNICODE_TO_GBK[20578] := 16#7364;
   // UNICODE_TO_GBK[20579] := 16#AA96;
   // UNICODE_TO_GBK[20580] := 16#7365;
   // UNICODE_TO_GBK[20581] := 16#AA97;
   // UNICODE_TO_GBK[20582] := 16#7366;
   // UNICODE_TO_GBK[20583] := 16#AA98;
   // UNICODE_TO_GBK[20584] := 16#7367;
   // UNICODE_TO_GBK[20585] := 16#AA99;
   // UNICODE_TO_GBK[20586] := 16#7368;
   // UNICODE_TO_GBK[20587] := 16#AA9A;
   // UNICODE_TO_GBK[20588] := 16#7369;
   // UNICODE_TO_GBK[20589] := 16#AA9B;
   // UNICODE_TO_GBK[20590] := 16#736A;
   // UNICODE_TO_GBK[20591] := 16#AA9C;
   // UNICODE_TO_GBK[20592] := 16#736B;
   // UNICODE_TO_GBK[20593] := 16#AA9D;
   // UNICODE_TO_GBK[20594] := 16#736C;
   // UNICODE_TO_GBK[20595] := 16#E2B3;
   // UNICODE_TO_GBK[20596] := 16#736D;
   // UNICODE_TO_GBK[20597] := 16#CCA1;
   // UNICODE_TO_GBK[20598] := 16#736E;
   // UNICODE_TO_GBK[20599] := 16#AA9E;
   // UNICODE_TO_GBK[20600] := 16#736F;
   // UNICODE_TO_GBK[20601] := 16#E2B4;
   // UNICODE_TO_GBK[20602] := 16#7370;
   // UNICODE_TO_GBK[20603] := 16#AA9F;
   // UNICODE_TO_GBK[20604] := 16#7371;
   // UNICODE_TO_GBK[20605] := 16#AAA0;
   // UNICODE_TO_GBK[20606] := 16#7372;
   // UNICODE_TO_GBK[20607] := 16#AB40;
   // UNICODE_TO_GBK[20608] := 16#7373;
   // UNICODE_TO_GBK[20609] := 16#AB41;
   // UNICODE_TO_GBK[20610] := 16#7374;
   // UNICODE_TO_GBK[20611] := 16#AB42;
   // UNICODE_TO_GBK[20612] := 16#7375;
   // UNICODE_TO_GBK[20613] := 16#AB43;
   // UNICODE_TO_GBK[20614] := 16#7376;
   // UNICODE_TO_GBK[20615] := 16#AB44;
   // UNICODE_TO_GBK[20616] := 16#7377;
   // UNICODE_TO_GBK[20617] := 16#AB45;
   // UNICODE_TO_GBK[20618] := 16#7378;
   // UNICODE_TO_GBK[20619] := 16#AB46;
   // UNICODE_TO_GBK[20620] := 16#7379;
   // UNICODE_TO_GBK[20621] := 16#AB47;
   // UNICODE_TO_GBK[20622] := 16#737A;
   // UNICODE_TO_GBK[20623] := 16#AB48;
   // UNICODE_TO_GBK[20624] := 16#737B;
   // UNICODE_TO_GBK[20625] := 16#AB49;
   // UNICODE_TO_GBK[20626] := 16#737C;
   // UNICODE_TO_GBK[20627] := 16#AB4A;
   // UNICODE_TO_GBK[20628] := 16#737D;
   // UNICODE_TO_GBK[20629] := 16#AB4B;
   // UNICODE_TO_GBK[20630] := 16#737E;
   // UNICODE_TO_GBK[20631] := 16#E2B5;
   // UNICODE_TO_GBK[20632] := 16#737F;
   // UNICODE_TO_GBK[20633] := 16#AB4C;
   // UNICODE_TO_GBK[20634] := 16#7380;
   // UNICODE_TO_GBK[20635] := 16#AB4D;
   // UNICODE_TO_GBK[20636] := 16#7381;
   // UNICODE_TO_GBK[20637] := 16#AB4E;
   // UNICODE_TO_GBK[20638] := 16#7382;
   // UNICODE_TO_GBK[20639] := 16#AB4F;
   // UNICODE_TO_GBK[20640] := 16#7383;
   // UNICODE_TO_GBK[20641] := 16#AB50;
   // UNICODE_TO_GBK[20642] := 16#7384;
   // UNICODE_TO_GBK[20643] := 16#D0FE;
   // UNICODE_TO_GBK[20644] := 16#7385;
   // UNICODE_TO_GBK[20645] := 16#AB51;
   // UNICODE_TO_GBK[20646] := 16#7386;
   // UNICODE_TO_GBK[20647] := 16#AB52;
   // UNICODE_TO_GBK[20648] := 16#7387;
   // UNICODE_TO_GBK[20649] := 16#C2CA;
   // UNICODE_TO_GBK[20650] := 16#7388;
   // UNICODE_TO_GBK[20651] := 16#AB53;
   // UNICODE_TO_GBK[20652] := 16#7389;
   // UNICODE_TO_GBK[20653] := 16#D3F1;
   // UNICODE_TO_GBK[20654] := 16#738A;
   // UNICODE_TO_GBK[20655] := 16#AB54;
   // UNICODE_TO_GBK[20656] := 16#738B;
   // UNICODE_TO_GBK[20657] := 16#CDF5;
   // UNICODE_TO_GBK[20658] := 16#738C;
   // UNICODE_TO_GBK[20659] := 16#AB55;
   // UNICODE_TO_GBK[20660] := 16#738D;
   // UNICODE_TO_GBK[20661] := 16#AB56;
   // UNICODE_TO_GBK[20662] := 16#738E;
   // UNICODE_TO_GBK[20663] := 16#E7E0;
   // UNICODE_TO_GBK[20664] := 16#738F;
   // UNICODE_TO_GBK[20665] := 16#AB57;
   // UNICODE_TO_GBK[20666] := 16#7390;
   // UNICODE_TO_GBK[20667] := 16#AB58;
   // UNICODE_TO_GBK[20668] := 16#7391;
   // UNICODE_TO_GBK[20669] := 16#E7E1;
   // UNICODE_TO_GBK[20670] := 16#7392;
   // UNICODE_TO_GBK[20671] := 16#AB59;
   // UNICODE_TO_GBK[20672] := 16#7393;
   // UNICODE_TO_GBK[20673] := 16#AB5A;
   // UNICODE_TO_GBK[20674] := 16#7394;
   // UNICODE_TO_GBK[20675] := 16#AB5B;
   // UNICODE_TO_GBK[20676] := 16#7395;
   // UNICODE_TO_GBK[20677] := 16#AB5C;
   // UNICODE_TO_GBK[20678] := 16#7396;
   // UNICODE_TO_GBK[20679] := 16#BEC1;
   // UNICODE_TO_GBK[20680] := 16#7397;
   // UNICODE_TO_GBK[20681] := 16#AB5D;
   // UNICODE_TO_GBK[20682] := 16#7398;
   // UNICODE_TO_GBK[20683] := 16#AB5E;
   // UNICODE_TO_GBK[20684] := 16#7399;
   // UNICODE_TO_GBK[20685] := 16#AB5F;
   // UNICODE_TO_GBK[20686] := 16#739A;
   // UNICODE_TO_GBK[20687] := 16#AB60;
   // UNICODE_TO_GBK[20688] := 16#739B;
   // UNICODE_TO_GBK[20689] := 16#C2EA;
   // UNICODE_TO_GBK[20690] := 16#739C;
   // UNICODE_TO_GBK[20691] := 16#AB61;
   // UNICODE_TO_GBK[20692] := 16#739D;
   // UNICODE_TO_GBK[20693] := 16#AB62;
   // UNICODE_TO_GBK[20694] := 16#739E;
   // UNICODE_TO_GBK[20695] := 16#AB63;
   // UNICODE_TO_GBK[20696] := 16#739F;
   // UNICODE_TO_GBK[20697] := 16#E7E4;
   // UNICODE_TO_GBK[20698] := 16#73A0;
   // UNICODE_TO_GBK[20699] := 16#AB64;
   // UNICODE_TO_GBK[20700] := 16#73A1;
   // UNICODE_TO_GBK[20701] := 16#AB65;
   // UNICODE_TO_GBK[20702] := 16#73A2;
   // UNICODE_TO_GBK[20703] := 16#E7E3;
   // UNICODE_TO_GBK[20704] := 16#73A3;
   // UNICODE_TO_GBK[20705] := 16#AB66;
   // UNICODE_TO_GBK[20706] := 16#73A4;
   // UNICODE_TO_GBK[20707] := 16#AB67;
   // UNICODE_TO_GBK[20708] := 16#73A5;
   // UNICODE_TO_GBK[20709] := 16#AB68;
   // UNICODE_TO_GBK[20710] := 16#73A6;
   // UNICODE_TO_GBK[20711] := 16#AB69;
   // UNICODE_TO_GBK[20712] := 16#73A7;
   // UNICODE_TO_GBK[20713] := 16#AB6A;
   // UNICODE_TO_GBK[20714] := 16#73A8;
   // UNICODE_TO_GBK[20715] := 16#AB6B;
   // UNICODE_TO_GBK[20716] := 16#73A9;
   // UNICODE_TO_GBK[20717] := 16#CDE6;
   // UNICODE_TO_GBK[20718] := 16#73AA;
   // UNICODE_TO_GBK[20719] := 16#AB6C;
   // UNICODE_TO_GBK[20720] := 16#73AB;
   // UNICODE_TO_GBK[20721] := 16#C3B5;
   // UNICODE_TO_GBK[20722] := 16#73AC;
   // UNICODE_TO_GBK[20723] := 16#AB6D;
   // UNICODE_TO_GBK[20724] := 16#73AD;
   // UNICODE_TO_GBK[20725] := 16#AB6E;
   // UNICODE_TO_GBK[20726] := 16#73AE;
   // UNICODE_TO_GBK[20727] := 16#E7E2;
   // UNICODE_TO_GBK[20728] := 16#73AF;
   // UNICODE_TO_GBK[20729] := 16#BBB7;
   // UNICODE_TO_GBK[20730] := 16#73B0;
   // UNICODE_TO_GBK[20731] := 16#CFD6;
   // UNICODE_TO_GBK[20732] := 16#73B1;
   // UNICODE_TO_GBK[20733] := 16#AB6F;
   // UNICODE_TO_GBK[20734] := 16#73B2;
   // UNICODE_TO_GBK[20735] := 16#C1E1;
   // UNICODE_TO_GBK[20736] := 16#73B3;
   // UNICODE_TO_GBK[20737] := 16#E7E9;
   // UNICODE_TO_GBK[20738] := 16#73B4;
   // UNICODE_TO_GBK[20739] := 16#AB70;
   // UNICODE_TO_GBK[20740] := 16#73B5;
   // UNICODE_TO_GBK[20741] := 16#AB71;
   // UNICODE_TO_GBK[20742] := 16#73B6;
   // UNICODE_TO_GBK[20743] := 16#AB72;
   // UNICODE_TO_GBK[20744] := 16#73B7;
   // UNICODE_TO_GBK[20745] := 16#E7E8;
   // UNICODE_TO_GBK[20746] := 16#73B8;
   // UNICODE_TO_GBK[20747] := 16#AB73;
   // UNICODE_TO_GBK[20748] := 16#73B9;
   // UNICODE_TO_GBK[20749] := 16#AB74;
   // UNICODE_TO_GBK[20750] := 16#73BA;
   // UNICODE_TO_GBK[20751] := 16#E7F4;
   // UNICODE_TO_GBK[20752] := 16#73BB;
   // UNICODE_TO_GBK[20753] := 16#B2A3;
   // UNICODE_TO_GBK[20754] := 16#73BC;
   // UNICODE_TO_GBK[20755] := 16#AB75;
   // UNICODE_TO_GBK[20756] := 16#73BD;
   // UNICODE_TO_GBK[20757] := 16#AB76;
   // UNICODE_TO_GBK[20758] := 16#73BE;
   // UNICODE_TO_GBK[20759] := 16#AB77;
   // UNICODE_TO_GBK[20760] := 16#73BF;
   // UNICODE_TO_GBK[20761] := 16#AB78;
   // UNICODE_TO_GBK[20762] := 16#73C0;
   // UNICODE_TO_GBK[20763] := 16#E7EA;
   // UNICODE_TO_GBK[20764] := 16#73C1;
   // UNICODE_TO_GBK[20765] := 16#AB79;
   // UNICODE_TO_GBK[20766] := 16#73C2;
   // UNICODE_TO_GBK[20767] := 16#E7E6;
   // UNICODE_TO_GBK[20768] := 16#73C3;
   // UNICODE_TO_GBK[20769] := 16#AB7A;
   // UNICODE_TO_GBK[20770] := 16#73C4;
   // UNICODE_TO_GBK[20771] := 16#AB7B;
   // UNICODE_TO_GBK[20772] := 16#73C5;
   // UNICODE_TO_GBK[20773] := 16#AB7C;
   // UNICODE_TO_GBK[20774] := 16#73C6;
   // UNICODE_TO_GBK[20775] := 16#AB7D;
   // UNICODE_TO_GBK[20776] := 16#73C7;
   // UNICODE_TO_GBK[20777] := 16#AB7E;
   // UNICODE_TO_GBK[20778] := 16#73C8;
   // UNICODE_TO_GBK[20779] := 16#E7EC;
   // UNICODE_TO_GBK[20780] := 16#73C9;
   // UNICODE_TO_GBK[20781] := 16#E7EB;
   // UNICODE_TO_GBK[20782] := 16#73CA;
   // UNICODE_TO_GBK[20783] := 16#C9BA;
   // UNICODE_TO_GBK[20784] := 16#73CB;
   // UNICODE_TO_GBK[20785] := 16#AB80;
   // UNICODE_TO_GBK[20786] := 16#73CC;
   // UNICODE_TO_GBK[20787] := 16#AB81;
   // UNICODE_TO_GBK[20788] := 16#73CD;
   // UNICODE_TO_GBK[20789] := 16#D5E4;
   // UNICODE_TO_GBK[20790] := 16#73CE;
   // UNICODE_TO_GBK[20791] := 16#AB82;
   // UNICODE_TO_GBK[20792] := 16#73CF;
   // UNICODE_TO_GBK[20793] := 16#E7E5;
   // UNICODE_TO_GBK[20794] := 16#73D0;
   // UNICODE_TO_GBK[20795] := 16#B7A9;
   // UNICODE_TO_GBK[20796] := 16#73D1;
   // UNICODE_TO_GBK[20797] := 16#E7E7;
   // UNICODE_TO_GBK[20798] := 16#73D2;
   // UNICODE_TO_GBK[20799] := 16#AB83;
   // UNICODE_TO_GBK[20800] := 16#73D3;
   // UNICODE_TO_GBK[20801] := 16#AB84;
   // UNICODE_TO_GBK[20802] := 16#73D4;
   // UNICODE_TO_GBK[20803] := 16#AB85;
   // UNICODE_TO_GBK[20804] := 16#73D5;
   // UNICODE_TO_GBK[20805] := 16#AB86;
   // UNICODE_TO_GBK[20806] := 16#73D6;
   // UNICODE_TO_GBK[20807] := 16#AB87;
   // UNICODE_TO_GBK[20808] := 16#73D7;
   // UNICODE_TO_GBK[20809] := 16#AB88;
   // UNICODE_TO_GBK[20810] := 16#73D8;
   // UNICODE_TO_GBK[20811] := 16#AB89;
   // UNICODE_TO_GBK[20812] := 16#73D9;
   // UNICODE_TO_GBK[20813] := 16#E7EE;
   // UNICODE_TO_GBK[20814] := 16#73DA;
   // UNICODE_TO_GBK[20815] := 16#AB8A;
   // UNICODE_TO_GBK[20816] := 16#73DB;
   // UNICODE_TO_GBK[20817] := 16#AB8B;
   // UNICODE_TO_GBK[20818] := 16#73DC;
   // UNICODE_TO_GBK[20819] := 16#AB8C;
   // UNICODE_TO_GBK[20820] := 16#73DD;
   // UNICODE_TO_GBK[20821] := 16#AB8D;
   // UNICODE_TO_GBK[20822] := 16#73DE;
   // UNICODE_TO_GBK[20823] := 16#E7F3;
   // UNICODE_TO_GBK[20824] := 16#73DF;
   // UNICODE_TO_GBK[20825] := 16#AB8E;
   // UNICODE_TO_GBK[20826] := 16#73E0;
   // UNICODE_TO_GBK[20827] := 16#D6E9;
   // UNICODE_TO_GBK[20828] := 16#73E1;
   // UNICODE_TO_GBK[20829] := 16#AB8F;
   // UNICODE_TO_GBK[20830] := 16#73E2;
   // UNICODE_TO_GBK[20831] := 16#AB90;
   // UNICODE_TO_GBK[20832] := 16#73E3;
   // UNICODE_TO_GBK[20833] := 16#AB91;
   // UNICODE_TO_GBK[20834] := 16#73E4;
   // UNICODE_TO_GBK[20835] := 16#AB92;
   // UNICODE_TO_GBK[20836] := 16#73E5;
   // UNICODE_TO_GBK[20837] := 16#E7ED;
   // UNICODE_TO_GBK[20838] := 16#73E6;
   // UNICODE_TO_GBK[20839] := 16#AB93;
   // UNICODE_TO_GBK[20840] := 16#73E7;
   // UNICODE_TO_GBK[20841] := 16#E7F2;
   // UNICODE_TO_GBK[20842] := 16#73E8;
   // UNICODE_TO_GBK[20843] := 16#AB94;
   // UNICODE_TO_GBK[20844] := 16#73E9;
   // UNICODE_TO_GBK[20845] := 16#E7F1;
   // UNICODE_TO_GBK[20846] := 16#73EA;
   // UNICODE_TO_GBK[20847] := 16#AB95;
   // UNICODE_TO_GBK[20848] := 16#73EB;
   // UNICODE_TO_GBK[20849] := 16#AB96;
   // UNICODE_TO_GBK[20850] := 16#73EC;
   // UNICODE_TO_GBK[20851] := 16#AB97;
   // UNICODE_TO_GBK[20852] := 16#73ED;
   // UNICODE_TO_GBK[20853] := 16#B0E0;
   // UNICODE_TO_GBK[20854] := 16#73EE;
   // UNICODE_TO_GBK[20855] := 16#AB98;
   // UNICODE_TO_GBK[20856] := 16#73EF;
   // UNICODE_TO_GBK[20857] := 16#AB99;
   // UNICODE_TO_GBK[20858] := 16#73F0;
   // UNICODE_TO_GBK[20859] := 16#AB9A;
   // UNICODE_TO_GBK[20860] := 16#73F1;
   // UNICODE_TO_GBK[20861] := 16#AB9B;
   // UNICODE_TO_GBK[20862] := 16#73F2;
   // UNICODE_TO_GBK[20863] := 16#E7F5;
   // UNICODE_TO_GBK[20864] := 16#73F3;
   // UNICODE_TO_GBK[20865] := 16#AB9C;
   // UNICODE_TO_GBK[20866] := 16#73F4;
   // UNICODE_TO_GBK[20867] := 16#AB9D;
   // UNICODE_TO_GBK[20868] := 16#73F5;
   // UNICODE_TO_GBK[20869] := 16#AB9E;
   // UNICODE_TO_GBK[20870] := 16#73F6;
   // UNICODE_TO_GBK[20871] := 16#AB9F;
   // UNICODE_TO_GBK[20872] := 16#73F7;
   // UNICODE_TO_GBK[20873] := 16#ABA0;
   // UNICODE_TO_GBK[20874] := 16#73F8;
   // UNICODE_TO_GBK[20875] := 16#AC40;
   // UNICODE_TO_GBK[20876] := 16#73F9;
   // UNICODE_TO_GBK[20877] := 16#AC41;
   // UNICODE_TO_GBK[20878] := 16#73FA;
   // UNICODE_TO_GBK[20879] := 16#AC42;
   // UNICODE_TO_GBK[20880] := 16#73FB;
   // UNICODE_TO_GBK[20881] := 16#AC43;
   // UNICODE_TO_GBK[20882] := 16#73FC;
   // UNICODE_TO_GBK[20883] := 16#AC44;
   // UNICODE_TO_GBK[20884] := 16#73FD;
   // UNICODE_TO_GBK[20885] := 16#AC45;
   // UNICODE_TO_GBK[20886] := 16#73FE;
   // UNICODE_TO_GBK[20887] := 16#AC46;
   // UNICODE_TO_GBK[20888] := 16#73FF;
   // UNICODE_TO_GBK[20889] := 16#AC47;
   // UNICODE_TO_GBK[20890] := 16#7400;
   // UNICODE_TO_GBK[20891] := 16#AC48;
   // UNICODE_TO_GBK[20892] := 16#7401;
   // UNICODE_TO_GBK[20893] := 16#AC49;
   // UNICODE_TO_GBK[20894] := 16#7402;
   // UNICODE_TO_GBK[20895] := 16#AC4A;
   // UNICODE_TO_GBK[20896] := 16#7403;
   // UNICODE_TO_GBK[20897] := 16#C7F2;
   // UNICODE_TO_GBK[20898] := 16#7404;
   // UNICODE_TO_GBK[20899] := 16#AC4B;
   // UNICODE_TO_GBK[20900] := 16#7405;
   // UNICODE_TO_GBK[20901] := 16#C0C5;
   // UNICODE_TO_GBK[20902] := 16#7406;
   // UNICODE_TO_GBK[20903] := 16#C0ED;
   // UNICODE_TO_GBK[20904] := 16#7407;
   // UNICODE_TO_GBK[20905] := 16#AC4C;
   // UNICODE_TO_GBK[20906] := 16#7408;
   // UNICODE_TO_GBK[20907] := 16#AC4D;
   // UNICODE_TO_GBK[20908] := 16#7409;
   // UNICODE_TO_GBK[20909] := 16#C1F0;
   // UNICODE_TO_GBK[20910] := 16#740A;
   // UNICODE_TO_GBK[20911] := 16#E7F0;
   // UNICODE_TO_GBK[20912] := 16#740B;
   // UNICODE_TO_GBK[20913] := 16#AC4E;
   // UNICODE_TO_GBK[20914] := 16#740C;
   // UNICODE_TO_GBK[20915] := 16#AC4F;
   // UNICODE_TO_GBK[20916] := 16#740D;
   // UNICODE_TO_GBK[20917] := 16#AC50;
   // UNICODE_TO_GBK[20918] := 16#740E;
   // UNICODE_TO_GBK[20919] := 16#AC51;
   // UNICODE_TO_GBK[20920] := 16#740F;
   // UNICODE_TO_GBK[20921] := 16#E7F6;
   // UNICODE_TO_GBK[20922] := 16#7410;
   // UNICODE_TO_GBK[20923] := 16#CBF6;
   // UNICODE_TO_GBK[20924] := 16#7411;
   // UNICODE_TO_GBK[20925] := 16#AC52;
   // UNICODE_TO_GBK[20926] := 16#7412;
   // UNICODE_TO_GBK[20927] := 16#AC53;
   // UNICODE_TO_GBK[20928] := 16#7413;
   // UNICODE_TO_GBK[20929] := 16#AC54;
   // UNICODE_TO_GBK[20930] := 16#7414;
   // UNICODE_TO_GBK[20931] := 16#AC55;
   // UNICODE_TO_GBK[20932] := 16#7415;
   // UNICODE_TO_GBK[20933] := 16#AC56;
   // UNICODE_TO_GBK[20934] := 16#7416;
   // UNICODE_TO_GBK[20935] := 16#AC57;
   // UNICODE_TO_GBK[20936] := 16#7417;
   // UNICODE_TO_GBK[20937] := 16#AC58;
   // UNICODE_TO_GBK[20938] := 16#7418;
   // UNICODE_TO_GBK[20939] := 16#AC59;
   // UNICODE_TO_GBK[20940] := 16#7419;
   // UNICODE_TO_GBK[20941] := 16#AC5A;
   // UNICODE_TO_GBK[20942] := 16#741A;
   // UNICODE_TO_GBK[20943] := 16#E8A2;
   // UNICODE_TO_GBK[20944] := 16#741B;
   // UNICODE_TO_GBK[20945] := 16#E8A1;
   // UNICODE_TO_GBK[20946] := 16#741C;
   // UNICODE_TO_GBK[20947] := 16#AC5B;
   // UNICODE_TO_GBK[20948] := 16#741D;
   // UNICODE_TO_GBK[20949] := 16#AC5C;
   // UNICODE_TO_GBK[20950] := 16#741E;
   // UNICODE_TO_GBK[20951] := 16#AC5D;
   // UNICODE_TO_GBK[20952] := 16#741F;
   // UNICODE_TO_GBK[20953] := 16#AC5E;
   // UNICODE_TO_GBK[20954] := 16#7420;
   // UNICODE_TO_GBK[20955] := 16#AC5F;
   // UNICODE_TO_GBK[20956] := 16#7421;
   // UNICODE_TO_GBK[20957] := 16#AC60;
   // UNICODE_TO_GBK[20958] := 16#7422;
   // UNICODE_TO_GBK[20959] := 16#D7C1;
   // UNICODE_TO_GBK[20960] := 16#7423;
   // UNICODE_TO_GBK[20961] := 16#AC61;
   // UNICODE_TO_GBK[20962] := 16#7424;
   // UNICODE_TO_GBK[20963] := 16#AC62;
   // UNICODE_TO_GBK[20964] := 16#7425;
   // UNICODE_TO_GBK[20965] := 16#E7FA;
   // UNICODE_TO_GBK[20966] := 16#7426;
   // UNICODE_TO_GBK[20967] := 16#E7F9;
   // UNICODE_TO_GBK[20968] := 16#7427;
   // UNICODE_TO_GBK[20969] := 16#AC63;
   // UNICODE_TO_GBK[20970] := 16#7428;
   // UNICODE_TO_GBK[20971] := 16#E7FB;
   // UNICODE_TO_GBK[20972] := 16#7429;
   // UNICODE_TO_GBK[20973] := 16#AC64;
   // UNICODE_TO_GBK[20974] := 16#742A;
   // UNICODE_TO_GBK[20975] := 16#E7F7;
   // UNICODE_TO_GBK[20976] := 16#742B;
   // UNICODE_TO_GBK[20977] := 16#AC65;
   // UNICODE_TO_GBK[20978] := 16#742C;
   // UNICODE_TO_GBK[20979] := 16#E7FE;
   // UNICODE_TO_GBK[20980] := 16#742D;
   // UNICODE_TO_GBK[20981] := 16#AC66;
   // UNICODE_TO_GBK[20982] := 16#742E;
   // UNICODE_TO_GBK[20983] := 16#E7FD;
   // UNICODE_TO_GBK[20984] := 16#742F;
   // UNICODE_TO_GBK[20985] := 16#AC67;
   // UNICODE_TO_GBK[20986] := 16#7430;
   // UNICODE_TO_GBK[20987] := 16#E7FC;
   // UNICODE_TO_GBK[20988] := 16#7431;
   // UNICODE_TO_GBK[20989] := 16#AC68;
   // UNICODE_TO_GBK[20990] := 16#7432;
   // UNICODE_TO_GBK[20991] := 16#AC69;
   // UNICODE_TO_GBK[20992] := 16#7433;
   // UNICODE_TO_GBK[20993] := 16#C1D5;
   // UNICODE_TO_GBK[20994] := 16#7434;
   // UNICODE_TO_GBK[20995] := 16#C7D9;
   // UNICODE_TO_GBK[20996] := 16#7435;
   // UNICODE_TO_GBK[20997] := 16#C5FD;
   // UNICODE_TO_GBK[20998] := 16#7436;
   // UNICODE_TO_GBK[20999] := 16#C5C3;
   // UNICODE_TO_GBK[21000] := 16#7437;
   // UNICODE_TO_GBK[21001] := 16#AC6A;
   // UNICODE_TO_GBK[21002] := 16#7438;
   // UNICODE_TO_GBK[21003] := 16#AC6B;
   // UNICODE_TO_GBK[21004] := 16#7439;
   // UNICODE_TO_GBK[21005] := 16#AC6C;
   // UNICODE_TO_GBK[21006] := 16#743A;
   // UNICODE_TO_GBK[21007] := 16#AC6D;
   // UNICODE_TO_GBK[21008] := 16#743B;
   // UNICODE_TO_GBK[21009] := 16#AC6E;
   // UNICODE_TO_GBK[21010] := 16#743C;
   // UNICODE_TO_GBK[21011] := 16#C7ED;
   // UNICODE_TO_GBK[21012] := 16#743D;
   // UNICODE_TO_GBK[21013] := 16#AC6F;
   // UNICODE_TO_GBK[21014] := 16#743E;
   // UNICODE_TO_GBK[21015] := 16#AC70;
   // UNICODE_TO_GBK[21016] := 16#743F;
   // UNICODE_TO_GBK[21017] := 16#AC71;
   // UNICODE_TO_GBK[21018] := 16#7440;
   // UNICODE_TO_GBK[21019] := 16#AC72;
   // UNICODE_TO_GBK[21020] := 16#7441;
   // UNICODE_TO_GBK[21021] := 16#E8A3;
   // UNICODE_TO_GBK[21022] := 16#7442;
   // UNICODE_TO_GBK[21023] := 16#AC73;
   // UNICODE_TO_GBK[21024] := 16#7443;
   // UNICODE_TO_GBK[21025] := 16#AC74;
   // UNICODE_TO_GBK[21026] := 16#7444;
   // UNICODE_TO_GBK[21027] := 16#AC75;
   // UNICODE_TO_GBK[21028] := 16#7445;
   // UNICODE_TO_GBK[21029] := 16#AC76;
   // UNICODE_TO_GBK[21030] := 16#7446;
   // UNICODE_TO_GBK[21031] := 16#AC77;
   // UNICODE_TO_GBK[21032] := 16#7447;
   // UNICODE_TO_GBK[21033] := 16#AC78;
   // UNICODE_TO_GBK[21034] := 16#7448;
   // UNICODE_TO_GBK[21035] := 16#AC79;
   // UNICODE_TO_GBK[21036] := 16#7449;
   // UNICODE_TO_GBK[21037] := 16#AC7A;
   // UNICODE_TO_GBK[21038] := 16#744A;
   // UNICODE_TO_GBK[21039] := 16#AC7B;
   // UNICODE_TO_GBK[21040] := 16#744B;
   // UNICODE_TO_GBK[21041] := 16#AC7C;
   // UNICODE_TO_GBK[21042] := 16#744C;
   // UNICODE_TO_GBK[21043] := 16#AC7D;
   // UNICODE_TO_GBK[21044] := 16#744D;
   // UNICODE_TO_GBK[21045] := 16#AC7E;
   // UNICODE_TO_GBK[21046] := 16#744E;
   // UNICODE_TO_GBK[21047] := 16#AC80;
   // UNICODE_TO_GBK[21048] := 16#744F;
   // UNICODE_TO_GBK[21049] := 16#AC81;
   // UNICODE_TO_GBK[21050] := 16#7450;
   // UNICODE_TO_GBK[21051] := 16#AC82;
   // UNICODE_TO_GBK[21052] := 16#7451;
   // UNICODE_TO_GBK[21053] := 16#AC83;
   // UNICODE_TO_GBK[21054] := 16#7452;
   // UNICODE_TO_GBK[21055] := 16#AC84;
   // UNICODE_TO_GBK[21056] := 16#7453;
   // UNICODE_TO_GBK[21057] := 16#AC85;
   // UNICODE_TO_GBK[21058] := 16#7454;
   // UNICODE_TO_GBK[21059] := 16#AC86;
   // UNICODE_TO_GBK[21060] := 16#7455;
   // UNICODE_TO_GBK[21061] := 16#E8A6;
   // UNICODE_TO_GBK[21062] := 16#7456;
   // UNICODE_TO_GBK[21063] := 16#AC87;
   // UNICODE_TO_GBK[21064] := 16#7457;
   // UNICODE_TO_GBK[21065] := 16#E8A5;
   // UNICODE_TO_GBK[21066] := 16#7458;
   // UNICODE_TO_GBK[21067] := 16#AC88;
   // UNICODE_TO_GBK[21068] := 16#7459;
   // UNICODE_TO_GBK[21069] := 16#E8A7;
   // UNICODE_TO_GBK[21070] := 16#745A;
   // UNICODE_TO_GBK[21071] := 16#BAF7;
   // UNICODE_TO_GBK[21072] := 16#745B;
   // UNICODE_TO_GBK[21073] := 16#E7F8;
   // UNICODE_TO_GBK[21074] := 16#745C;
   // UNICODE_TO_GBK[21075] := 16#E8A4;
   // UNICODE_TO_GBK[21076] := 16#745D;
   // UNICODE_TO_GBK[21077] := 16#AC89;
   // UNICODE_TO_GBK[21078] := 16#745E;
   // UNICODE_TO_GBK[21079] := 16#C8F0;
   // UNICODE_TO_GBK[21080] := 16#745F;
   // UNICODE_TO_GBK[21081] := 16#C9AA;
   // UNICODE_TO_GBK[21082] := 16#7460;
   // UNICODE_TO_GBK[21083] := 16#AC8A;
   // UNICODE_TO_GBK[21084] := 16#7461;
   // UNICODE_TO_GBK[21085] := 16#AC8B;
   // UNICODE_TO_GBK[21086] := 16#7462;
   // UNICODE_TO_GBK[21087] := 16#AC8C;
   // UNICODE_TO_GBK[21088] := 16#7463;
   // UNICODE_TO_GBK[21089] := 16#AC8D;
   // UNICODE_TO_GBK[21090] := 16#7464;
   // UNICODE_TO_GBK[21091] := 16#AC8E;
   // UNICODE_TO_GBK[21092] := 16#7465;
   // UNICODE_TO_GBK[21093] := 16#AC8F;
   // UNICODE_TO_GBK[21094] := 16#7466;
   // UNICODE_TO_GBK[21095] := 16#AC90;
   // UNICODE_TO_GBK[21096] := 16#7467;
   // UNICODE_TO_GBK[21097] := 16#AC91;
   // UNICODE_TO_GBK[21098] := 16#7468;
   // UNICODE_TO_GBK[21099] := 16#AC92;
   // UNICODE_TO_GBK[21100] := 16#7469;
   // UNICODE_TO_GBK[21101] := 16#AC93;
   // UNICODE_TO_GBK[21102] := 16#746A;
   // UNICODE_TO_GBK[21103] := 16#AC94;
   // UNICODE_TO_GBK[21104] := 16#746B;
   // UNICODE_TO_GBK[21105] := 16#AC95;
   // UNICODE_TO_GBK[21106] := 16#746C;
   // UNICODE_TO_GBK[21107] := 16#AC96;
   // UNICODE_TO_GBK[21108] := 16#746D;
   // UNICODE_TO_GBK[21109] := 16#E8A9;
   // UNICODE_TO_GBK[21110] := 16#746E;
   // UNICODE_TO_GBK[21111] := 16#AC97;
   // UNICODE_TO_GBK[21112] := 16#746F;
   // UNICODE_TO_GBK[21113] := 16#AC98;
   // UNICODE_TO_GBK[21114] := 16#7470;
   // UNICODE_TO_GBK[21115] := 16#B9E5;
   // UNICODE_TO_GBK[21116] := 16#7471;
   // UNICODE_TO_GBK[21117] := 16#AC99;
   // UNICODE_TO_GBK[21118] := 16#7472;
   // UNICODE_TO_GBK[21119] := 16#AC9A;
   // UNICODE_TO_GBK[21120] := 16#7473;
   // UNICODE_TO_GBK[21121] := 16#AC9B;
   // UNICODE_TO_GBK[21122] := 16#7474;
   // UNICODE_TO_GBK[21123] := 16#AC9C;
   // UNICODE_TO_GBK[21124] := 16#7475;
   // UNICODE_TO_GBK[21125] := 16#AC9D;
   // UNICODE_TO_GBK[21126] := 16#7476;
   // UNICODE_TO_GBK[21127] := 16#D1FE;
   // UNICODE_TO_GBK[21128] := 16#7477;
   // UNICODE_TO_GBK[21129] := 16#E8A8;
   // UNICODE_TO_GBK[21130] := 16#7478;
   // UNICODE_TO_GBK[21131] := 16#AC9E;
   // UNICODE_TO_GBK[21132] := 16#7479;
   // UNICODE_TO_GBK[21133] := 16#AC9F;
   // UNICODE_TO_GBK[21134] := 16#747A;
   // UNICODE_TO_GBK[21135] := 16#ACA0;
   // UNICODE_TO_GBK[21136] := 16#747B;
   // UNICODE_TO_GBK[21137] := 16#AD40;
   // UNICODE_TO_GBK[21138] := 16#747C;
   // UNICODE_TO_GBK[21139] := 16#AD41;
   // UNICODE_TO_GBK[21140] := 16#747D;
   // UNICODE_TO_GBK[21141] := 16#AD42;
   // UNICODE_TO_GBK[21142] := 16#747E;
   // UNICODE_TO_GBK[21143] := 16#E8AA;
   // UNICODE_TO_GBK[21144] := 16#747F;
   // UNICODE_TO_GBK[21145] := 16#AD43;
   // UNICODE_TO_GBK[21146] := 16#7480;
   // UNICODE_TO_GBK[21147] := 16#E8AD;
   // UNICODE_TO_GBK[21148] := 16#7481;
   // UNICODE_TO_GBK[21149] := 16#E8AE;
   // UNICODE_TO_GBK[21150] := 16#7482;
   // UNICODE_TO_GBK[21151] := 16#AD44;
   // UNICODE_TO_GBK[21152] := 16#7483;
   // UNICODE_TO_GBK[21153] := 16#C1A7;
   // UNICODE_TO_GBK[21154] := 16#7484;
   // UNICODE_TO_GBK[21155] := 16#AD45;
   // UNICODE_TO_GBK[21156] := 16#7485;
   // UNICODE_TO_GBK[21157] := 16#AD46;
   // UNICODE_TO_GBK[21158] := 16#7486;
   // UNICODE_TO_GBK[21159] := 16#AD47;
   // UNICODE_TO_GBK[21160] := 16#7487;
   // UNICODE_TO_GBK[21161] := 16#E8AF;
   // UNICODE_TO_GBK[21162] := 16#7488;
   // UNICODE_TO_GBK[21163] := 16#AD48;
   // UNICODE_TO_GBK[21164] := 16#7489;
   // UNICODE_TO_GBK[21165] := 16#AD49;
   // UNICODE_TO_GBK[21166] := 16#748A;
   // UNICODE_TO_GBK[21167] := 16#AD4A;
   // UNICODE_TO_GBK[21168] := 16#748B;
   // UNICODE_TO_GBK[21169] := 16#E8B0;
   // UNICODE_TO_GBK[21170] := 16#748C;
   // UNICODE_TO_GBK[21171] := 16#AD4B;
   // UNICODE_TO_GBK[21172] := 16#748D;
   // UNICODE_TO_GBK[21173] := 16#AD4C;
   // UNICODE_TO_GBK[21174] := 16#748E;
   // UNICODE_TO_GBK[21175] := 16#E8AC;
   // UNICODE_TO_GBK[21176] := 16#748F;
   // UNICODE_TO_GBK[21177] := 16#AD4D;
   // UNICODE_TO_GBK[21178] := 16#7490;
   // UNICODE_TO_GBK[21179] := 16#E8B4;
   // UNICODE_TO_GBK[21180] := 16#7491;
   // UNICODE_TO_GBK[21181] := 16#AD4E;
   // UNICODE_TO_GBK[21182] := 16#7492;
   // UNICODE_TO_GBK[21183] := 16#AD4F;
   // UNICODE_TO_GBK[21184] := 16#7493;
   // UNICODE_TO_GBK[21185] := 16#AD50;
   // UNICODE_TO_GBK[21186] := 16#7494;
   // UNICODE_TO_GBK[21187] := 16#AD51;
   // UNICODE_TO_GBK[21188] := 16#7495;
   // UNICODE_TO_GBK[21189] := 16#AD52;
   // UNICODE_TO_GBK[21190] := 16#7496;
   // UNICODE_TO_GBK[21191] := 16#AD53;
   // UNICODE_TO_GBK[21192] := 16#7497;
   // UNICODE_TO_GBK[21193] := 16#AD54;
   // UNICODE_TO_GBK[21194] := 16#7498;
   // UNICODE_TO_GBK[21195] := 16#AD55;
   // UNICODE_TO_GBK[21196] := 16#7499;
   // UNICODE_TO_GBK[21197] := 16#AD56;
   // UNICODE_TO_GBK[21198] := 16#749A;
   // UNICODE_TO_GBK[21199] := 16#AD57;
   // UNICODE_TO_GBK[21200] := 16#749B;
   // UNICODE_TO_GBK[21201] := 16#AD58;
   // UNICODE_TO_GBK[21202] := 16#749C;
   // UNICODE_TO_GBK[21203] := 16#E8AB;
   // UNICODE_TO_GBK[21204] := 16#749D;
   // UNICODE_TO_GBK[21205] := 16#AD59;
   // UNICODE_TO_GBK[21206] := 16#749E;
   // UNICODE_TO_GBK[21207] := 16#E8B1;
   // UNICODE_TO_GBK[21208] := 16#749F;
   // UNICODE_TO_GBK[21209] := 16#AD5A;
   // UNICODE_TO_GBK[21210] := 16#74A0;
   // UNICODE_TO_GBK[21211] := 16#AD5B;
   // UNICODE_TO_GBK[21212] := 16#74A1;
   // UNICODE_TO_GBK[21213] := 16#AD5C;
   // UNICODE_TO_GBK[21214] := 16#74A2;
   // UNICODE_TO_GBK[21215] := 16#AD5D;
   // UNICODE_TO_GBK[21216] := 16#74A3;
   // UNICODE_TO_GBK[21217] := 16#AD5E;
   // UNICODE_TO_GBK[21218] := 16#74A4;
   // UNICODE_TO_GBK[21219] := 16#AD5F;
   // UNICODE_TO_GBK[21220] := 16#74A5;
   // UNICODE_TO_GBK[21221] := 16#AD60;
   // UNICODE_TO_GBK[21222] := 16#74A6;
   // UNICODE_TO_GBK[21223] := 16#AD61;
   // UNICODE_TO_GBK[21224] := 16#74A7;
   // UNICODE_TO_GBK[21225] := 16#E8B5;
   // UNICODE_TO_GBK[21226] := 16#74A8;
   // UNICODE_TO_GBK[21227] := 16#E8B2;
   // UNICODE_TO_GBK[21228] := 16#74A9;
   // UNICODE_TO_GBK[21229] := 16#E8B3;
   // UNICODE_TO_GBK[21230] := 16#74AA;
   // UNICODE_TO_GBK[21231] := 16#AD62;
   // UNICODE_TO_GBK[21232] := 16#74AB;
   // UNICODE_TO_GBK[21233] := 16#AD63;
   // UNICODE_TO_GBK[21234] := 16#74AC;
   // UNICODE_TO_GBK[21235] := 16#AD64;
   // UNICODE_TO_GBK[21236] := 16#74AD;
   // UNICODE_TO_GBK[21237] := 16#AD65;
   // UNICODE_TO_GBK[21238] := 16#74AE;
   // UNICODE_TO_GBK[21239] := 16#AD66;
   // UNICODE_TO_GBK[21240] := 16#74AF;
   // UNICODE_TO_GBK[21241] := 16#AD67;
   // UNICODE_TO_GBK[21242] := 16#74B0;
   // UNICODE_TO_GBK[21243] := 16#AD68;
   // UNICODE_TO_GBK[21244] := 16#74B1;
   // UNICODE_TO_GBK[21245] := 16#AD69;
   // UNICODE_TO_GBK[21246] := 16#74B2;
   // UNICODE_TO_GBK[21247] := 16#AD6A;
   // UNICODE_TO_GBK[21248] := 16#74B3;
   // UNICODE_TO_GBK[21249] := 16#AD6B;
   // UNICODE_TO_GBK[21250] := 16#74B4;
   // UNICODE_TO_GBK[21251] := 16#AD6C;
   // UNICODE_TO_GBK[21252] := 16#74B5;
   // UNICODE_TO_GBK[21253] := 16#AD6D;
   // UNICODE_TO_GBK[21254] := 16#74B6;
   // UNICODE_TO_GBK[21255] := 16#AD6E;
   // UNICODE_TO_GBK[21256] := 16#74B7;
   // UNICODE_TO_GBK[21257] := 16#AD6F;
   // UNICODE_TO_GBK[21258] := 16#74B8;
   // UNICODE_TO_GBK[21259] := 16#AD70;
   // UNICODE_TO_GBK[21260] := 16#74B9;
   // UNICODE_TO_GBK[21261] := 16#AD71;
   // UNICODE_TO_GBK[21262] := 16#74BA;
   // UNICODE_TO_GBK[21263] := 16#E8B7;
   // UNICODE_TO_GBK[21264] := 16#74BB;
   // UNICODE_TO_GBK[21265] := 16#AD72;
   // UNICODE_TO_GBK[21266] := 16#74BC;
   // UNICODE_TO_GBK[21267] := 16#AD73;
   // UNICODE_TO_GBK[21268] := 16#74BD;
   // UNICODE_TO_GBK[21269] := 16#AD74;
   // UNICODE_TO_GBK[21270] := 16#74BE;
   // UNICODE_TO_GBK[21271] := 16#AD75;
   // UNICODE_TO_GBK[21272] := 16#74BF;
   // UNICODE_TO_GBK[21273] := 16#AD76;
   // UNICODE_TO_GBK[21274] := 16#74C0;
   // UNICODE_TO_GBK[21275] := 16#AD77;
   // UNICODE_TO_GBK[21276] := 16#74C1;
   // UNICODE_TO_GBK[21277] := 16#AD78;
   // UNICODE_TO_GBK[21278] := 16#74C2;
   // UNICODE_TO_GBK[21279] := 16#AD79;
   // UNICODE_TO_GBK[21280] := 16#74C3;
   // UNICODE_TO_GBK[21281] := 16#AD7A;
   // UNICODE_TO_GBK[21282] := 16#74C4;
   // UNICODE_TO_GBK[21283] := 16#AD7B;
   // UNICODE_TO_GBK[21284] := 16#74C5;
   // UNICODE_TO_GBK[21285] := 16#AD7C;
   // UNICODE_TO_GBK[21286] := 16#74C6;
   // UNICODE_TO_GBK[21287] := 16#AD7D;
   // UNICODE_TO_GBK[21288] := 16#74C7;
   // UNICODE_TO_GBK[21289] := 16#AD7E;
   // UNICODE_TO_GBK[21290] := 16#74C8;
   // UNICODE_TO_GBK[21291] := 16#AD80;
   // UNICODE_TO_GBK[21292] := 16#74C9;
   // UNICODE_TO_GBK[21293] := 16#AD81;
   // UNICODE_TO_GBK[21294] := 16#74CA;
   // UNICODE_TO_GBK[21295] := 16#AD82;
   // UNICODE_TO_GBK[21296] := 16#74CB;
   // UNICODE_TO_GBK[21297] := 16#AD83;
   // UNICODE_TO_GBK[21298] := 16#74CC;
   // UNICODE_TO_GBK[21299] := 16#AD84;
   // UNICODE_TO_GBK[21300] := 16#74CD;
   // UNICODE_TO_GBK[21301] := 16#AD85;
   // UNICODE_TO_GBK[21302] := 16#74CE;
   // UNICODE_TO_GBK[21303] := 16#AD86;
   // UNICODE_TO_GBK[21304] := 16#74CF;
   // UNICODE_TO_GBK[21305] := 16#AD87;
   // UNICODE_TO_GBK[21306] := 16#74D0;
   // UNICODE_TO_GBK[21307] := 16#AD88;
   // UNICODE_TO_GBK[21308] := 16#74D1;
   // UNICODE_TO_GBK[21309] := 16#AD89;
   // UNICODE_TO_GBK[21310] := 16#74D2;
   // UNICODE_TO_GBK[21311] := 16#E8B6;
   // UNICODE_TO_GBK[21312] := 16#74D3;
   // UNICODE_TO_GBK[21313] := 16#AD8A;
   // UNICODE_TO_GBK[21314] := 16#74D4;
   // UNICODE_TO_GBK[21315] := 16#AD8B;
   // UNICODE_TO_GBK[21316] := 16#74D5;
   // UNICODE_TO_GBK[21317] := 16#AD8C;
   // UNICODE_TO_GBK[21318] := 16#74D6;
   // UNICODE_TO_GBK[21319] := 16#AD8D;
   // UNICODE_TO_GBK[21320] := 16#74D7;
   // UNICODE_TO_GBK[21321] := 16#AD8E;
   // UNICODE_TO_GBK[21322] := 16#74D8;
   // UNICODE_TO_GBK[21323] := 16#AD8F;
   // UNICODE_TO_GBK[21324] := 16#74D9;
   // UNICODE_TO_GBK[21325] := 16#AD90;
   // UNICODE_TO_GBK[21326] := 16#74DA;
   // UNICODE_TO_GBK[21327] := 16#AD91;
   // UNICODE_TO_GBK[21328] := 16#74DB;
   // UNICODE_TO_GBK[21329] := 16#AD92;
   // UNICODE_TO_GBK[21330] := 16#74DC;
   // UNICODE_TO_GBK[21331] := 16#B9CF;
   // UNICODE_TO_GBK[21332] := 16#74DD;
   // UNICODE_TO_GBK[21333] := 16#AD93;
   // UNICODE_TO_GBK[21334] := 16#74DE;
   // UNICODE_TO_GBK[21335] := 16#F0AC;
   // UNICODE_TO_GBK[21336] := 16#74DF;
   // UNICODE_TO_GBK[21337] := 16#AD94;
   // UNICODE_TO_GBK[21338] := 16#74E0;
   // UNICODE_TO_GBK[21339] := 16#F0AD;
   // UNICODE_TO_GBK[21340] := 16#74E1;
   // UNICODE_TO_GBK[21341] := 16#AD95;
   // UNICODE_TO_GBK[21342] := 16#74E2;
   // UNICODE_TO_GBK[21343] := 16#C6B0;
   // UNICODE_TO_GBK[21344] := 16#74E3;
   // UNICODE_TO_GBK[21345] := 16#B0EA;
   // UNICODE_TO_GBK[21346] := 16#74E4;
   // UNICODE_TO_GBK[21347] := 16#C8BF;
   // UNICODE_TO_GBK[21348] := 16#74E5;
   // UNICODE_TO_GBK[21349] := 16#AD96;
   // UNICODE_TO_GBK[21350] := 16#74E6;
   // UNICODE_TO_GBK[21351] := 16#CDDF;
   // UNICODE_TO_GBK[21352] := 16#74E7;
   // UNICODE_TO_GBK[21353] := 16#AD97;
   // UNICODE_TO_GBK[21354] := 16#74E8;
   // UNICODE_TO_GBK[21355] := 16#AD98;
   // UNICODE_TO_GBK[21356] := 16#74E9;
   // UNICODE_TO_GBK[21357] := 16#AD99;
   // UNICODE_TO_GBK[21358] := 16#74EA;
   // UNICODE_TO_GBK[21359] := 16#AD9A;
   // UNICODE_TO_GBK[21360] := 16#74EB;
   // UNICODE_TO_GBK[21361] := 16#AD9B;
   // UNICODE_TO_GBK[21362] := 16#74EC;
   // UNICODE_TO_GBK[21363] := 16#AD9C;
   // UNICODE_TO_GBK[21364] := 16#74ED;
   // UNICODE_TO_GBK[21365] := 16#AD9D;
   // UNICODE_TO_GBK[21366] := 16#74EE;
   // UNICODE_TO_GBK[21367] := 16#CECD;
   // UNICODE_TO_GBK[21368] := 16#74EF;
   // UNICODE_TO_GBK[21369] := 16#EAB1;
   // UNICODE_TO_GBK[21370] := 16#74F0;
   // UNICODE_TO_GBK[21371] := 16#AD9E;
   // UNICODE_TO_GBK[21372] := 16#74F1;
   // UNICODE_TO_GBK[21373] := 16#AD9F;
   // UNICODE_TO_GBK[21374] := 16#74F2;
   // UNICODE_TO_GBK[21375] := 16#ADA0;
   // UNICODE_TO_GBK[21376] := 16#74F3;
   // UNICODE_TO_GBK[21377] := 16#AE40;
   // UNICODE_TO_GBK[21378] := 16#74F4;
   // UNICODE_TO_GBK[21379] := 16#EAB2;
   // UNICODE_TO_GBK[21380] := 16#74F5;
   // UNICODE_TO_GBK[21381] := 16#AE41;
   // UNICODE_TO_GBK[21382] := 16#74F6;
   // UNICODE_TO_GBK[21383] := 16#C6BF;
   // UNICODE_TO_GBK[21384] := 16#74F7;
   // UNICODE_TO_GBK[21385] := 16#B4C9;
   // UNICODE_TO_GBK[21386] := 16#74F8;
   // UNICODE_TO_GBK[21387] := 16#AE42;
   // UNICODE_TO_GBK[21388] := 16#74F9;
   // UNICODE_TO_GBK[21389] := 16#AE43;
   // UNICODE_TO_GBK[21390] := 16#74FA;
   // UNICODE_TO_GBK[21391] := 16#AE44;
   // UNICODE_TO_GBK[21392] := 16#74FB;
   // UNICODE_TO_GBK[21393] := 16#AE45;
   // UNICODE_TO_GBK[21394] := 16#74FC;
   // UNICODE_TO_GBK[21395] := 16#AE46;
   // UNICODE_TO_GBK[21396] := 16#74FD;
   // UNICODE_TO_GBK[21397] := 16#AE47;
   // UNICODE_TO_GBK[21398] := 16#74FE;
   // UNICODE_TO_GBK[21399] := 16#AE48;
   // UNICODE_TO_GBK[21400] := 16#74FF;
   // UNICODE_TO_GBK[21401] := 16#EAB3;
   // UNICODE_TO_GBK[21402] := 16#7500;
   // UNICODE_TO_GBK[21403] := 16#AE49;
   // UNICODE_TO_GBK[21404] := 16#7501;
   // UNICODE_TO_GBK[21405] := 16#AE4A;
   // UNICODE_TO_GBK[21406] := 16#7502;
   // UNICODE_TO_GBK[21407] := 16#AE4B;
   // UNICODE_TO_GBK[21408] := 16#7503;
   // UNICODE_TO_GBK[21409] := 16#AE4C;
   // UNICODE_TO_GBK[21410] := 16#7504;
   // UNICODE_TO_GBK[21411] := 16#D5E7;
   // UNICODE_TO_GBK[21412] := 16#7505;
   // UNICODE_TO_GBK[21413] := 16#AE4D;
   // UNICODE_TO_GBK[21414] := 16#7506;
   // UNICODE_TO_GBK[21415] := 16#AE4E;
   // UNICODE_TO_GBK[21416] := 16#7507;
   // UNICODE_TO_GBK[21417] := 16#AE4F;
   // UNICODE_TO_GBK[21418] := 16#7508;
   // UNICODE_TO_GBK[21419] := 16#AE50;
   // UNICODE_TO_GBK[21420] := 16#7509;
   // UNICODE_TO_GBK[21421] := 16#AE51;
   // UNICODE_TO_GBK[21422] := 16#750A;
   // UNICODE_TO_GBK[21423] := 16#AE52;
   // UNICODE_TO_GBK[21424] := 16#750B;
   // UNICODE_TO_GBK[21425] := 16#AE53;
   // UNICODE_TO_GBK[21426] := 16#750C;
   // UNICODE_TO_GBK[21427] := 16#AE54;
   // UNICODE_TO_GBK[21428] := 16#750D;
   // UNICODE_TO_GBK[21429] := 16#DDF9;
   // UNICODE_TO_GBK[21430] := 16#750E;
   // UNICODE_TO_GBK[21431] := 16#AE55;
   // UNICODE_TO_GBK[21432] := 16#750F;
   // UNICODE_TO_GBK[21433] := 16#EAB4;
   // UNICODE_TO_GBK[21434] := 16#7510;
   // UNICODE_TO_GBK[21435] := 16#AE56;
   // UNICODE_TO_GBK[21436] := 16#7511;
   // UNICODE_TO_GBK[21437] := 16#EAB5;
   // UNICODE_TO_GBK[21438] := 16#7512;
   // UNICODE_TO_GBK[21439] := 16#AE57;
   // UNICODE_TO_GBK[21440] := 16#7513;
   // UNICODE_TO_GBK[21441] := 16#EAB6;
   // UNICODE_TO_GBK[21442] := 16#7514;
   // UNICODE_TO_GBK[21443] := 16#AE58;
   // UNICODE_TO_GBK[21444] := 16#7515;
   // UNICODE_TO_GBK[21445] := 16#AE59;
   // UNICODE_TO_GBK[21446] := 16#7516;
   // UNICODE_TO_GBK[21447] := 16#AE5A;
   // UNICODE_TO_GBK[21448] := 16#7517;
   // UNICODE_TO_GBK[21449] := 16#AE5B;
   // UNICODE_TO_GBK[21450] := 16#7518;
   // UNICODE_TO_GBK[21451] := 16#B8CA;
   // UNICODE_TO_GBK[21452] := 16#7519;
   // UNICODE_TO_GBK[21453] := 16#DFB0;
   // UNICODE_TO_GBK[21454] := 16#751A;
   // UNICODE_TO_GBK[21455] := 16#C9F5;
   // UNICODE_TO_GBK[21456] := 16#751B;
   // UNICODE_TO_GBK[21457] := 16#AE5C;
   // UNICODE_TO_GBK[21458] := 16#751C;
   // UNICODE_TO_GBK[21459] := 16#CCF0;
   // UNICODE_TO_GBK[21460] := 16#751D;
   // UNICODE_TO_GBK[21461] := 16#AE5D;
   // UNICODE_TO_GBK[21462] := 16#751E;
   // UNICODE_TO_GBK[21463] := 16#AE5E;
   // UNICODE_TO_GBK[21464] := 16#751F;
   // UNICODE_TO_GBK[21465] := 16#C9FA;
   // UNICODE_TO_GBK[21466] := 16#7520;
   // UNICODE_TO_GBK[21467] := 16#AE5F;
   // UNICODE_TO_GBK[21468] := 16#7521;
   // UNICODE_TO_GBK[21469] := 16#AE60;
   // UNICODE_TO_GBK[21470] := 16#7522;
   // UNICODE_TO_GBK[21471] := 16#AE61;
   // UNICODE_TO_GBK[21472] := 16#7523;
   // UNICODE_TO_GBK[21473] := 16#AE62;
   // UNICODE_TO_GBK[21474] := 16#7524;
   // UNICODE_TO_GBK[21475] := 16#AE63;
   // UNICODE_TO_GBK[21476] := 16#7525;
   // UNICODE_TO_GBK[21477] := 16#C9FB;
   // UNICODE_TO_GBK[21478] := 16#7526;
   // UNICODE_TO_GBK[21479] := 16#AE64;
   // UNICODE_TO_GBK[21480] := 16#7527;
   // UNICODE_TO_GBK[21481] := 16#AE65;
   // UNICODE_TO_GBK[21482] := 16#7528;
   // UNICODE_TO_GBK[21483] := 16#D3C3;
   // UNICODE_TO_GBK[21484] := 16#7529;
   // UNICODE_TO_GBK[21485] := 16#CBA6;
   // UNICODE_TO_GBK[21486] := 16#752A;
   // UNICODE_TO_GBK[21487] := 16#AE66;
   // UNICODE_TO_GBK[21488] := 16#752B;
   // UNICODE_TO_GBK[21489] := 16#B8A6;
   // UNICODE_TO_GBK[21490] := 16#752C;
   // UNICODE_TO_GBK[21491] := 16#F0AE;
   // UNICODE_TO_GBK[21492] := 16#752D;
   // UNICODE_TO_GBK[21493] := 16#B1C2;
   // UNICODE_TO_GBK[21494] := 16#752E;
   // UNICODE_TO_GBK[21495] := 16#AE67;
   // UNICODE_TO_GBK[21496] := 16#752F;
   // UNICODE_TO_GBK[21497] := 16#E5B8;
   // UNICODE_TO_GBK[21498] := 16#7530;
   // UNICODE_TO_GBK[21499] := 16#CCEF;
   // UNICODE_TO_GBK[21500] := 16#7531;
   // UNICODE_TO_GBK[21501] := 16#D3C9;
   // UNICODE_TO_GBK[21502] := 16#7532;
   // UNICODE_TO_GBK[21503] := 16#BCD7;
   // UNICODE_TO_GBK[21504] := 16#7533;
   // UNICODE_TO_GBK[21505] := 16#C9EA;
   // UNICODE_TO_GBK[21506] := 16#7534;
   // UNICODE_TO_GBK[21507] := 16#AE68;
   // UNICODE_TO_GBK[21508] := 16#7535;
   // UNICODE_TO_GBK[21509] := 16#B5E7;
   // UNICODE_TO_GBK[21510] := 16#7536;
   // UNICODE_TO_GBK[21511] := 16#AE69;
   // UNICODE_TO_GBK[21512] := 16#7537;
   // UNICODE_TO_GBK[21513] := 16#C4D0;
   // UNICODE_TO_GBK[21514] := 16#7538;
   // UNICODE_TO_GBK[21515] := 16#B5E9;
   // UNICODE_TO_GBK[21516] := 16#7539;
   // UNICODE_TO_GBK[21517] := 16#AE6A;
   // UNICODE_TO_GBK[21518] := 16#753A;
   // UNICODE_TO_GBK[21519] := 16#EEAE;
   // UNICODE_TO_GBK[21520] := 16#753B;
   // UNICODE_TO_GBK[21521] := 16#BBAD;
   // UNICODE_TO_GBK[21522] := 16#753C;
   // UNICODE_TO_GBK[21523] := 16#AE6B;
   // UNICODE_TO_GBK[21524] := 16#753D;
   // UNICODE_TO_GBK[21525] := 16#AE6C;
   // UNICODE_TO_GBK[21526] := 16#753E;
   // UNICODE_TO_GBK[21527] := 16#E7DE;
   // UNICODE_TO_GBK[21528] := 16#753F;
   // UNICODE_TO_GBK[21529] := 16#AE6D;
   // UNICODE_TO_GBK[21530] := 16#7540;
   // UNICODE_TO_GBK[21531] := 16#EEAF;
   // UNICODE_TO_GBK[21532] := 16#7541;
   // UNICODE_TO_GBK[21533] := 16#AE6E;
   // UNICODE_TO_GBK[21534] := 16#7542;
   // UNICODE_TO_GBK[21535] := 16#AE6F;
   // UNICODE_TO_GBK[21536] := 16#7543;
   // UNICODE_TO_GBK[21537] := 16#AE70;
   // UNICODE_TO_GBK[21538] := 16#7544;
   // UNICODE_TO_GBK[21539] := 16#AE71;
   // UNICODE_TO_GBK[21540] := 16#7545;
   // UNICODE_TO_GBK[21541] := 16#B3A9;
   // UNICODE_TO_GBK[21542] := 16#7546;
   // UNICODE_TO_GBK[21543] := 16#AE72;
   // UNICODE_TO_GBK[21544] := 16#7547;
   // UNICODE_TO_GBK[21545] := 16#AE73;
   // UNICODE_TO_GBK[21546] := 16#7548;
   // UNICODE_TO_GBK[21547] := 16#EEB2;
   // UNICODE_TO_GBK[21548] := 16#7549;
   // UNICODE_TO_GBK[21549] := 16#AE74;
   // UNICODE_TO_GBK[21550] := 16#754A;
   // UNICODE_TO_GBK[21551] := 16#AE75;
   // UNICODE_TO_GBK[21552] := 16#754B;
   // UNICODE_TO_GBK[21553] := 16#EEB1;
   // UNICODE_TO_GBK[21554] := 16#754C;
   // UNICODE_TO_GBK[21555] := 16#BDE7;
   // UNICODE_TO_GBK[21556] := 16#754D;
   // UNICODE_TO_GBK[21557] := 16#AE76;
   // UNICODE_TO_GBK[21558] := 16#754E;
   // UNICODE_TO_GBK[21559] := 16#EEB0;
   // UNICODE_TO_GBK[21560] := 16#754F;
   // UNICODE_TO_GBK[21561] := 16#CEB7;
   // UNICODE_TO_GBK[21562] := 16#7550;
   // UNICODE_TO_GBK[21563] := 16#AE77;
   // UNICODE_TO_GBK[21564] := 16#7551;
   // UNICODE_TO_GBK[21565] := 16#AE78;
   // UNICODE_TO_GBK[21566] := 16#7552;
   // UNICODE_TO_GBK[21567] := 16#AE79;
   // UNICODE_TO_GBK[21568] := 16#7553;
   // UNICODE_TO_GBK[21569] := 16#AE7A;
   // UNICODE_TO_GBK[21570] := 16#7554;
   // UNICODE_TO_GBK[21571] := 16#C5CF;
   // UNICODE_TO_GBK[21572] := 16#7555;
   // UNICODE_TO_GBK[21573] := 16#AE7B;
   // UNICODE_TO_GBK[21574] := 16#7556;
   // UNICODE_TO_GBK[21575] := 16#AE7C;
   // UNICODE_TO_GBK[21576] := 16#7557;
   // UNICODE_TO_GBK[21577] := 16#AE7D;
   // UNICODE_TO_GBK[21578] := 16#7558;
   // UNICODE_TO_GBK[21579] := 16#AE7E;
   // UNICODE_TO_GBK[21580] := 16#7559;
   // UNICODE_TO_GBK[21581] := 16#C1F4;
   // UNICODE_TO_GBK[21582] := 16#755A;
   // UNICODE_TO_GBK[21583] := 16#DBCE;
   // UNICODE_TO_GBK[21584] := 16#755B;
   // UNICODE_TO_GBK[21585] := 16#EEB3;
   // UNICODE_TO_GBK[21586] := 16#755C;
   // UNICODE_TO_GBK[21587] := 16#D0F3;
   // UNICODE_TO_GBK[21588] := 16#755D;
   // UNICODE_TO_GBK[21589] := 16#AE80;
   // UNICODE_TO_GBK[21590] := 16#755E;
   // UNICODE_TO_GBK[21591] := 16#AE81;
   // UNICODE_TO_GBK[21592] := 16#755F;
   // UNICODE_TO_GBK[21593] := 16#AE82;
   // UNICODE_TO_GBK[21594] := 16#7560;
   // UNICODE_TO_GBK[21595] := 16#AE83;
   // UNICODE_TO_GBK[21596] := 16#7561;
   // UNICODE_TO_GBK[21597] := 16#AE84;
   // UNICODE_TO_GBK[21598] := 16#7562;
   // UNICODE_TO_GBK[21599] := 16#AE85;
   // UNICODE_TO_GBK[21600] := 16#7563;
   // UNICODE_TO_GBK[21601] := 16#AE86;
   // UNICODE_TO_GBK[21602] := 16#7564;
   // UNICODE_TO_GBK[21603] := 16#AE87;
   // UNICODE_TO_GBK[21604] := 16#7565;
   // UNICODE_TO_GBK[21605] := 16#C2D4;
   // UNICODE_TO_GBK[21606] := 16#7566;
   // UNICODE_TO_GBK[21607] := 16#C6E8;
   // UNICODE_TO_GBK[21608] := 16#7567;
   // UNICODE_TO_GBK[21609] := 16#AE88;
   // UNICODE_TO_GBK[21610] := 16#7568;
   // UNICODE_TO_GBK[21611] := 16#AE89;
   // UNICODE_TO_GBK[21612] := 16#7569;
   // UNICODE_TO_GBK[21613] := 16#AE8A;
   // UNICODE_TO_GBK[21614] := 16#756A;
   // UNICODE_TO_GBK[21615] := 16#B7AC;
   // UNICODE_TO_GBK[21616] := 16#756B;
   // UNICODE_TO_GBK[21617] := 16#AE8B;
   // UNICODE_TO_GBK[21618] := 16#756C;
   // UNICODE_TO_GBK[21619] := 16#AE8C;
   // UNICODE_TO_GBK[21620] := 16#756D;
   // UNICODE_TO_GBK[21621] := 16#AE8D;
   // UNICODE_TO_GBK[21622] := 16#756E;
   // UNICODE_TO_GBK[21623] := 16#AE8E;
   // UNICODE_TO_GBK[21624] := 16#756F;
   // UNICODE_TO_GBK[21625] := 16#AE8F;
   // UNICODE_TO_GBK[21626] := 16#7570;
   // UNICODE_TO_GBK[21627] := 16#AE90;
   // UNICODE_TO_GBK[21628] := 16#7571;
   // UNICODE_TO_GBK[21629] := 16#AE91;
   // UNICODE_TO_GBK[21630] := 16#7572;
   // UNICODE_TO_GBK[21631] := 16#EEB4;
   // UNICODE_TO_GBK[21632] := 16#7573;
   // UNICODE_TO_GBK[21633] := 16#AE92;
   // UNICODE_TO_GBK[21634] := 16#7574;
   // UNICODE_TO_GBK[21635] := 16#B3EB;
   // UNICODE_TO_GBK[21636] := 16#7575;
   // UNICODE_TO_GBK[21637] := 16#AE93;
   // UNICODE_TO_GBK[21638] := 16#7576;
   // UNICODE_TO_GBK[21639] := 16#AE94;
   // UNICODE_TO_GBK[21640] := 16#7577;
   // UNICODE_TO_GBK[21641] := 16#AE95;
   // UNICODE_TO_GBK[21642] := 16#7578;
   // UNICODE_TO_GBK[21643] := 16#BBFB;
   // UNICODE_TO_GBK[21644] := 16#7579;
   // UNICODE_TO_GBK[21645] := 16#EEB5;
   // UNICODE_TO_GBK[21646] := 16#757A;
   // UNICODE_TO_GBK[21647] := 16#AE96;
   // UNICODE_TO_GBK[21648] := 16#757B;
   // UNICODE_TO_GBK[21649] := 16#AE97;
   // UNICODE_TO_GBK[21650] := 16#757C;
   // UNICODE_TO_GBK[21651] := 16#AE98;
   // UNICODE_TO_GBK[21652] := 16#757D;
   // UNICODE_TO_GBK[21653] := 16#AE99;
   // UNICODE_TO_GBK[21654] := 16#757E;
   // UNICODE_TO_GBK[21655] := 16#AE9A;
   // UNICODE_TO_GBK[21656] := 16#757F;
   // UNICODE_TO_GBK[21657] := 16#E7DC;
   // UNICODE_TO_GBK[21658] := 16#7580;
   // UNICODE_TO_GBK[21659] := 16#AE9B;
   // UNICODE_TO_GBK[21660] := 16#7581;
   // UNICODE_TO_GBK[21661] := 16#AE9C;
   // UNICODE_TO_GBK[21662] := 16#7582;
   // UNICODE_TO_GBK[21663] := 16#AE9D;
   // UNICODE_TO_GBK[21664] := 16#7583;
   // UNICODE_TO_GBK[21665] := 16#EEB6;
   // UNICODE_TO_GBK[21666] := 16#7584;
   // UNICODE_TO_GBK[21667] := 16#AE9E;
   // UNICODE_TO_GBK[21668] := 16#7585;
   // UNICODE_TO_GBK[21669] := 16#AE9F;
   // UNICODE_TO_GBK[21670] := 16#7586;
   // UNICODE_TO_GBK[21671] := 16#BDAE;
   // UNICODE_TO_GBK[21672] := 16#7587;
   // UNICODE_TO_GBK[21673] := 16#AEA0;
   // UNICODE_TO_GBK[21674] := 16#7588;
   // UNICODE_TO_GBK[21675] := 16#AF40;
   // UNICODE_TO_GBK[21676] := 16#7589;
   // UNICODE_TO_GBK[21677] := 16#AF41;
   // UNICODE_TO_GBK[21678] := 16#758A;
   // UNICODE_TO_GBK[21679] := 16#AF42;
   // UNICODE_TO_GBK[21680] := 16#758B;
   // UNICODE_TO_GBK[21681] := 16#F1E2;
   // UNICODE_TO_GBK[21682] := 16#758C;
   // UNICODE_TO_GBK[21683] := 16#AF43;
   // UNICODE_TO_GBK[21684] := 16#758D;
   // UNICODE_TO_GBK[21685] := 16#AF44;
   // UNICODE_TO_GBK[21686] := 16#758E;
   // UNICODE_TO_GBK[21687] := 16#AF45;
   // UNICODE_TO_GBK[21688] := 16#758F;
   // UNICODE_TO_GBK[21689] := 16#CAE8;
   // UNICODE_TO_GBK[21690] := 16#7590;
   // UNICODE_TO_GBK[21691] := 16#AF46;
   // UNICODE_TO_GBK[21692] := 16#7591;
   // UNICODE_TO_GBK[21693] := 16#D2C9;
   // UNICODE_TO_GBK[21694] := 16#7592;
   // UNICODE_TO_GBK[21695] := 16#F0DA;
   // UNICODE_TO_GBK[21696] := 16#7593;
   // UNICODE_TO_GBK[21697] := 16#AF47;
   // UNICODE_TO_GBK[21698] := 16#7594;
   // UNICODE_TO_GBK[21699] := 16#F0DB;
   // UNICODE_TO_GBK[21700] := 16#7595;
   // UNICODE_TO_GBK[21701] := 16#AF48;
   // UNICODE_TO_GBK[21702] := 16#7596;
   // UNICODE_TO_GBK[21703] := 16#F0DC;
   // UNICODE_TO_GBK[21704] := 16#7597;
   // UNICODE_TO_GBK[21705] := 16#C1C6;
   // UNICODE_TO_GBK[21706] := 16#7598;
   // UNICODE_TO_GBK[21707] := 16#AF49;
   // UNICODE_TO_GBK[21708] := 16#7599;
   // UNICODE_TO_GBK[21709] := 16#B8ED;
   // UNICODE_TO_GBK[21710] := 16#759A;
   // UNICODE_TO_GBK[21711] := 16#BECE;
   // UNICODE_TO_GBK[21712] := 16#759B;
   // UNICODE_TO_GBK[21713] := 16#AF4A;
   // UNICODE_TO_GBK[21714] := 16#759C;
   // UNICODE_TO_GBK[21715] := 16#AF4B;
   // UNICODE_TO_GBK[21716] := 16#759D;
   // UNICODE_TO_GBK[21717] := 16#F0DE;
   // UNICODE_TO_GBK[21718] := 16#759E;
   // UNICODE_TO_GBK[21719] := 16#AF4C;
   // UNICODE_TO_GBK[21720] := 16#759F;
   // UNICODE_TO_GBK[21721] := 16#C5B1;
   // UNICODE_TO_GBK[21722] := 16#75A0;
   // UNICODE_TO_GBK[21723] := 16#F0DD;
   // UNICODE_TO_GBK[21724] := 16#75A1;
   // UNICODE_TO_GBK[21725] := 16#D1F1;
   // UNICODE_TO_GBK[21726] := 16#75A2;
   // UNICODE_TO_GBK[21727] := 16#AF4D;
   // UNICODE_TO_GBK[21728] := 16#75A3;
   // UNICODE_TO_GBK[21729] := 16#F0E0;
   // UNICODE_TO_GBK[21730] := 16#75A4;
   // UNICODE_TO_GBK[21731] := 16#B0CC;
   // UNICODE_TO_GBK[21732] := 16#75A5;
   // UNICODE_TO_GBK[21733] := 16#BDEA;
   // UNICODE_TO_GBK[21734] := 16#75A6;
   // UNICODE_TO_GBK[21735] := 16#AF4E;
   // UNICODE_TO_GBK[21736] := 16#75A7;
   // UNICODE_TO_GBK[21737] := 16#AF4F;
   // UNICODE_TO_GBK[21738] := 16#75A8;
   // UNICODE_TO_GBK[21739] := 16#AF50;
   // UNICODE_TO_GBK[21740] := 16#75A9;
   // UNICODE_TO_GBK[21741] := 16#AF51;
   // UNICODE_TO_GBK[21742] := 16#75AA;
   // UNICODE_TO_GBK[21743] := 16#AF52;
   // UNICODE_TO_GBK[21744] := 16#75AB;
   // UNICODE_TO_GBK[21745] := 16#D2DF;
   // UNICODE_TO_GBK[21746] := 16#75AC;
   // UNICODE_TO_GBK[21747] := 16#F0DF;
   // UNICODE_TO_GBK[21748] := 16#75AD;
   // UNICODE_TO_GBK[21749] := 16#AF53;
   // UNICODE_TO_GBK[21750] := 16#75AE;
   // UNICODE_TO_GBK[21751] := 16#B4AF;
   // UNICODE_TO_GBK[21752] := 16#75AF;
   // UNICODE_TO_GBK[21753] := 16#B7E8;
   // UNICODE_TO_GBK[21754] := 16#75B0;
   // UNICODE_TO_GBK[21755] := 16#F0E6;
   // UNICODE_TO_GBK[21756] := 16#75B1;
   // UNICODE_TO_GBK[21757] := 16#F0E5;
   // UNICODE_TO_GBK[21758] := 16#75B2;
   // UNICODE_TO_GBK[21759] := 16#C6A3;
   // UNICODE_TO_GBK[21760] := 16#75B3;
   // UNICODE_TO_GBK[21761] := 16#F0E1;
   // UNICODE_TO_GBK[21762] := 16#75B4;
   // UNICODE_TO_GBK[21763] := 16#F0E2;
   // UNICODE_TO_GBK[21764] := 16#75B5;
   // UNICODE_TO_GBK[21765] := 16#B4C3;
   // UNICODE_TO_GBK[21766] := 16#75B6;
   // UNICODE_TO_GBK[21767] := 16#AF54;
   // UNICODE_TO_GBK[21768] := 16#75B7;
   // UNICODE_TO_GBK[21769] := 16#AF55;
   // UNICODE_TO_GBK[21770] := 16#75B8;
   // UNICODE_TO_GBK[21771] := 16#F0E3;
   // UNICODE_TO_GBK[21772] := 16#75B9;
   // UNICODE_TO_GBK[21773] := 16#D5EE;
   // UNICODE_TO_GBK[21774] := 16#75BA;
   // UNICODE_TO_GBK[21775] := 16#AF56;
   // UNICODE_TO_GBK[21776] := 16#75BB;
   // UNICODE_TO_GBK[21777] := 16#AF57;
   // UNICODE_TO_GBK[21778] := 16#75BC;
   // UNICODE_TO_GBK[21779] := 16#CCDB;
   // UNICODE_TO_GBK[21780] := 16#75BD;
   // UNICODE_TO_GBK[21781] := 16#BED2;
   // UNICODE_TO_GBK[21782] := 16#75BE;
   // UNICODE_TO_GBK[21783] := 16#BCB2;
   // UNICODE_TO_GBK[21784] := 16#75BF;
   // UNICODE_TO_GBK[21785] := 16#AF58;
   // UNICODE_TO_GBK[21786] := 16#75C0;
   // UNICODE_TO_GBK[21787] := 16#AF59;
   // UNICODE_TO_GBK[21788] := 16#75C1;
   // UNICODE_TO_GBK[21789] := 16#AF5A;
   // UNICODE_TO_GBK[21790] := 16#75C2;
   // UNICODE_TO_GBK[21791] := 16#F0E8;
   // UNICODE_TO_GBK[21792] := 16#75C3;
   // UNICODE_TO_GBK[21793] := 16#F0E7;
   // UNICODE_TO_GBK[21794] := 16#75C4;
   // UNICODE_TO_GBK[21795] := 16#F0E4;
   // UNICODE_TO_GBK[21796] := 16#75C5;
   // UNICODE_TO_GBK[21797] := 16#B2A1;
   // UNICODE_TO_GBK[21798] := 16#75C6;
   // UNICODE_TO_GBK[21799] := 16#AF5B;
   // UNICODE_TO_GBK[21800] := 16#75C7;
   // UNICODE_TO_GBK[21801] := 16#D6A2;
   // UNICODE_TO_GBK[21802] := 16#75C8;
   // UNICODE_TO_GBK[21803] := 16#D3B8;
   // UNICODE_TO_GBK[21804] := 16#75C9;
   // UNICODE_TO_GBK[21805] := 16#BEB7;
   // UNICODE_TO_GBK[21806] := 16#75CA;
   // UNICODE_TO_GBK[21807] := 16#C8AC;
   // UNICODE_TO_GBK[21808] := 16#75CB;
   // UNICODE_TO_GBK[21809] := 16#AF5C;
   // UNICODE_TO_GBK[21810] := 16#75CC;
   // UNICODE_TO_GBK[21811] := 16#AF5D;
   // UNICODE_TO_GBK[21812] := 16#75CD;
   // UNICODE_TO_GBK[21813] := 16#F0EA;
   // UNICODE_TO_GBK[21814] := 16#75CE;
   // UNICODE_TO_GBK[21815] := 16#AF5E;
   // UNICODE_TO_GBK[21816] := 16#75CF;
   // UNICODE_TO_GBK[21817] := 16#AF5F;
   // UNICODE_TO_GBK[21818] := 16#75D0;
   // UNICODE_TO_GBK[21819] := 16#AF60;
   // UNICODE_TO_GBK[21820] := 16#75D1;
   // UNICODE_TO_GBK[21821] := 16#AF61;
   // UNICODE_TO_GBK[21822] := 16#75D2;
   // UNICODE_TO_GBK[21823] := 16#D1F7;
   // UNICODE_TO_GBK[21824] := 16#75D3;
   // UNICODE_TO_GBK[21825] := 16#AF62;
   // UNICODE_TO_GBK[21826] := 16#75D4;
   // UNICODE_TO_GBK[21827] := 16#D6CC;
   // UNICODE_TO_GBK[21828] := 16#75D5;
   // UNICODE_TO_GBK[21829] := 16#BADB;
   // UNICODE_TO_GBK[21830] := 16#75D6;
   // UNICODE_TO_GBK[21831] := 16#F0E9;
   // UNICODE_TO_GBK[21832] := 16#75D7;
   // UNICODE_TO_GBK[21833] := 16#AF63;
   // UNICODE_TO_GBK[21834] := 16#75D8;
   // UNICODE_TO_GBK[21835] := 16#B6BB;
   // UNICODE_TO_GBK[21836] := 16#75D9;
   // UNICODE_TO_GBK[21837] := 16#AF64;
   // UNICODE_TO_GBK[21838] := 16#75DA;
   // UNICODE_TO_GBK[21839] := 16#AF65;
   // UNICODE_TO_GBK[21840] := 16#75DB;
   // UNICODE_TO_GBK[21841] := 16#CDB4;
   // UNICODE_TO_GBK[21842] := 16#75DC;
   // UNICODE_TO_GBK[21843] := 16#AF66;
   // UNICODE_TO_GBK[21844] := 16#75DD;
   // UNICODE_TO_GBK[21845] := 16#AF67;
   // UNICODE_TO_GBK[21846] := 16#75DE;
   // UNICODE_TO_GBK[21847] := 16#C6A6;
   // UNICODE_TO_GBK[21848] := 16#75DF;
   // UNICODE_TO_GBK[21849] := 16#AF68;
   // UNICODE_TO_GBK[21850] := 16#75E0;
   // UNICODE_TO_GBK[21851] := 16#AF69;
   // UNICODE_TO_GBK[21852] := 16#75E1;
   // UNICODE_TO_GBK[21853] := 16#AF6A;
   // UNICODE_TO_GBK[21854] := 16#75E2;
   // UNICODE_TO_GBK[21855] := 16#C1A1;
   // UNICODE_TO_GBK[21856] := 16#75E3;
   // UNICODE_TO_GBK[21857] := 16#F0EB;
   // UNICODE_TO_GBK[21858] := 16#75E4;
   // UNICODE_TO_GBK[21859] := 16#F0EE;
   // UNICODE_TO_GBK[21860] := 16#75E5;
   // UNICODE_TO_GBK[21861] := 16#AF6B;
   // UNICODE_TO_GBK[21862] := 16#75E6;
   // UNICODE_TO_GBK[21863] := 16#F0ED;
   // UNICODE_TO_GBK[21864] := 16#75E7;
   // UNICODE_TO_GBK[21865] := 16#F0F0;
   // UNICODE_TO_GBK[21866] := 16#75E8;
   // UNICODE_TO_GBK[21867] := 16#F0EC;
   // UNICODE_TO_GBK[21868] := 16#75E9;
   // UNICODE_TO_GBK[21869] := 16#AF6C;
   // UNICODE_TO_GBK[21870] := 16#75EA;
   // UNICODE_TO_GBK[21871] := 16#BBBE;
   // UNICODE_TO_GBK[21872] := 16#75EB;
   // UNICODE_TO_GBK[21873] := 16#F0EF;
   // UNICODE_TO_GBK[21874] := 16#75EC;
   // UNICODE_TO_GBK[21875] := 16#AF6D;
   // UNICODE_TO_GBK[21876] := 16#75ED;
   // UNICODE_TO_GBK[21877] := 16#AF6E;
   // UNICODE_TO_GBK[21878] := 16#75EE;
   // UNICODE_TO_GBK[21879] := 16#AF6F;
   // UNICODE_TO_GBK[21880] := 16#75EF;
   // UNICODE_TO_GBK[21881] := 16#AF70;
   // UNICODE_TO_GBK[21882] := 16#75F0;
   // UNICODE_TO_GBK[21883] := 16#CCB5;
   // UNICODE_TO_GBK[21884] := 16#75F1;
   // UNICODE_TO_GBK[21885] := 16#F0F2;
   // UNICODE_TO_GBK[21886] := 16#75F2;
   // UNICODE_TO_GBK[21887] := 16#AF71;
   // UNICODE_TO_GBK[21888] := 16#75F3;
   // UNICODE_TO_GBK[21889] := 16#AF72;
   // UNICODE_TO_GBK[21890] := 16#75F4;
   // UNICODE_TO_GBK[21891] := 16#B3D5;
   // UNICODE_TO_GBK[21892] := 16#75F5;
   // UNICODE_TO_GBK[21893] := 16#AF73;
   // UNICODE_TO_GBK[21894] := 16#75F6;
   // UNICODE_TO_GBK[21895] := 16#AF74;
   // UNICODE_TO_GBK[21896] := 16#75F7;
   // UNICODE_TO_GBK[21897] := 16#AF75;
   // UNICODE_TO_GBK[21898] := 16#75F8;
   // UNICODE_TO_GBK[21899] := 16#AF76;
   // UNICODE_TO_GBK[21900] := 16#75F9;
   // UNICODE_TO_GBK[21901] := 16#B1D4;
   // UNICODE_TO_GBK[21902] := 16#75FA;
   // UNICODE_TO_GBK[21903] := 16#AF77;
   // UNICODE_TO_GBK[21904] := 16#75FB;
   // UNICODE_TO_GBK[21905] := 16#AF78;
   // UNICODE_TO_GBK[21906] := 16#75FC;
   // UNICODE_TO_GBK[21907] := 16#F0F3;
   // UNICODE_TO_GBK[21908] := 16#75FD;
   // UNICODE_TO_GBK[21909] := 16#AF79;
   // UNICODE_TO_GBK[21910] := 16#75FE;
   // UNICODE_TO_GBK[21911] := 16#AF7A;
   // UNICODE_TO_GBK[21912] := 16#75FF;
   // UNICODE_TO_GBK[21913] := 16#F0F4;
   // UNICODE_TO_GBK[21914] := 16#7600;
   // UNICODE_TO_GBK[21915] := 16#F0F6;
   // UNICODE_TO_GBK[21916] := 16#7601;
   // UNICODE_TO_GBK[21917] := 16#B4E1;
   // UNICODE_TO_GBK[21918] := 16#7602;
   // UNICODE_TO_GBK[21919] := 16#AF7B;
   // UNICODE_TO_GBK[21920] := 16#7603;
   // UNICODE_TO_GBK[21921] := 16#F0F1;
   // UNICODE_TO_GBK[21922] := 16#7604;
   // UNICODE_TO_GBK[21923] := 16#AF7C;
   // UNICODE_TO_GBK[21924] := 16#7605;
   // UNICODE_TO_GBK[21925] := 16#F0F7;
   // UNICODE_TO_GBK[21926] := 16#7606;
   // UNICODE_TO_GBK[21927] := 16#AF7D;
   // UNICODE_TO_GBK[21928] := 16#7607;
   // UNICODE_TO_GBK[21929] := 16#AF7E;
   // UNICODE_TO_GBK[21930] := 16#7608;
   // UNICODE_TO_GBK[21931] := 16#AF80;
   // UNICODE_TO_GBK[21932] := 16#7609;
   // UNICODE_TO_GBK[21933] := 16#AF81;
   // UNICODE_TO_GBK[21934] := 16#760A;
   // UNICODE_TO_GBK[21935] := 16#F0FA;
   // UNICODE_TO_GBK[21936] := 16#760B;
   // UNICODE_TO_GBK[21937] := 16#AF82;
   // UNICODE_TO_GBK[21938] := 16#760C;
   // UNICODE_TO_GBK[21939] := 16#F0F8;
   // UNICODE_TO_GBK[21940] := 16#760D;
   // UNICODE_TO_GBK[21941] := 16#AF83;
   // UNICODE_TO_GBK[21942] := 16#760E;
   // UNICODE_TO_GBK[21943] := 16#AF84;
   // UNICODE_TO_GBK[21944] := 16#760F;
   // UNICODE_TO_GBK[21945] := 16#AF85;
   // UNICODE_TO_GBK[21946] := 16#7610;
   // UNICODE_TO_GBK[21947] := 16#F0F5;
   // UNICODE_TO_GBK[21948] := 16#7611;
   // UNICODE_TO_GBK[21949] := 16#AF86;
   // UNICODE_TO_GBK[21950] := 16#7612;
   // UNICODE_TO_GBK[21951] := 16#AF87;
   // UNICODE_TO_GBK[21952] := 16#7613;
   // UNICODE_TO_GBK[21953] := 16#AF88;
   // UNICODE_TO_GBK[21954] := 16#7614;
   // UNICODE_TO_GBK[21955] := 16#AF89;
   // UNICODE_TO_GBK[21956] := 16#7615;
   // UNICODE_TO_GBK[21957] := 16#F0FD;
   // UNICODE_TO_GBK[21958] := 16#7616;
   // UNICODE_TO_GBK[21959] := 16#AF8A;
   // UNICODE_TO_GBK[21960] := 16#7617;
   // UNICODE_TO_GBK[21961] := 16#F0F9;
   // UNICODE_TO_GBK[21962] := 16#7618;
   // UNICODE_TO_GBK[21963] := 16#F0FC;
   // UNICODE_TO_GBK[21964] := 16#7619;
   // UNICODE_TO_GBK[21965] := 16#F0FE;
   // UNICODE_TO_GBK[21966] := 16#761A;
   // UNICODE_TO_GBK[21967] := 16#AF8B;
   // UNICODE_TO_GBK[21968] := 16#761B;
   // UNICODE_TO_GBK[21969] := 16#F1A1;
   // UNICODE_TO_GBK[21970] := 16#761C;
   // UNICODE_TO_GBK[21971] := 16#AF8C;
   // UNICODE_TO_GBK[21972] := 16#761D;
   // UNICODE_TO_GBK[21973] := 16#AF8D;
   // UNICODE_TO_GBK[21974] := 16#761E;
   // UNICODE_TO_GBK[21975] := 16#AF8E;
   // UNICODE_TO_GBK[21976] := 16#761F;
   // UNICODE_TO_GBK[21977] := 16#CEC1;
   // UNICODE_TO_GBK[21978] := 16#7620;
   // UNICODE_TO_GBK[21979] := 16#F1A4;
   // UNICODE_TO_GBK[21980] := 16#7621;
   // UNICODE_TO_GBK[21981] := 16#AF8F;
   // UNICODE_TO_GBK[21982] := 16#7622;
   // UNICODE_TO_GBK[21983] := 16#F1A3;
   // UNICODE_TO_GBK[21984] := 16#7623;
   // UNICODE_TO_GBK[21985] := 16#AF90;
   // UNICODE_TO_GBK[21986] := 16#7624;
   // UNICODE_TO_GBK[21987] := 16#C1F6;
   // UNICODE_TO_GBK[21988] := 16#7625;
   // UNICODE_TO_GBK[21989] := 16#F0FB;
   // UNICODE_TO_GBK[21990] := 16#7626;
   // UNICODE_TO_GBK[21991] := 16#CADD;
   // UNICODE_TO_GBK[21992] := 16#7627;
   // UNICODE_TO_GBK[21993] := 16#AF91;
   // UNICODE_TO_GBK[21994] := 16#7628;
   // UNICODE_TO_GBK[21995] := 16#AF92;
   // UNICODE_TO_GBK[21996] := 16#7629;
   // UNICODE_TO_GBK[21997] := 16#B4F1;
   // UNICODE_TO_GBK[21998] := 16#762A;
   // UNICODE_TO_GBK[21999] := 16#B1F1;
   // UNICODE_TO_GBK[22000] := 16#762B;
   // UNICODE_TO_GBK[22001] := 16#CCB1;
   // UNICODE_TO_GBK[22002] := 16#762C;
   // UNICODE_TO_GBK[22003] := 16#AF93;
   // UNICODE_TO_GBK[22004] := 16#762D;
   // UNICODE_TO_GBK[22005] := 16#F1A6;
   // UNICODE_TO_GBK[22006] := 16#762E;
   // UNICODE_TO_GBK[22007] := 16#AF94;
   // UNICODE_TO_GBK[22008] := 16#762F;
   // UNICODE_TO_GBK[22009] := 16#AF95;
   // UNICODE_TO_GBK[22010] := 16#7630;
   // UNICODE_TO_GBK[22011] := 16#F1A7;
   // UNICODE_TO_GBK[22012] := 16#7631;
   // UNICODE_TO_GBK[22013] := 16#AF96;
   // UNICODE_TO_GBK[22014] := 16#7632;
   // UNICODE_TO_GBK[22015] := 16#AF97;
   // UNICODE_TO_GBK[22016] := 16#7633;
   // UNICODE_TO_GBK[22017] := 16#F1AC;
   // UNICODE_TO_GBK[22018] := 16#7634;
   // UNICODE_TO_GBK[22019] := 16#D5CE;
   // UNICODE_TO_GBK[22020] := 16#7635;
   // UNICODE_TO_GBK[22021] := 16#F1A9;
   // UNICODE_TO_GBK[22022] := 16#7636;
   // UNICODE_TO_GBK[22023] := 16#AF98;
   // UNICODE_TO_GBK[22024] := 16#7637;
   // UNICODE_TO_GBK[22025] := 16#AF99;
   // UNICODE_TO_GBK[22026] := 16#7638;
   // UNICODE_TO_GBK[22027] := 16#C8B3;
   // UNICODE_TO_GBK[22028] := 16#7639;
   // UNICODE_TO_GBK[22029] := 16#AF9A;
   // UNICODE_TO_GBK[22030] := 16#763A;
   // UNICODE_TO_GBK[22031] := 16#AF9B;
   // UNICODE_TO_GBK[22032] := 16#763B;
   // UNICODE_TO_GBK[22033] := 16#AF9C;
   // UNICODE_TO_GBK[22034] := 16#763C;
   // UNICODE_TO_GBK[22035] := 16#F1A2;
   // UNICODE_TO_GBK[22036] := 16#763D;
   // UNICODE_TO_GBK[22037] := 16#AF9D;
   // UNICODE_TO_GBK[22038] := 16#763E;
   // UNICODE_TO_GBK[22039] := 16#F1AB;
   // UNICODE_TO_GBK[22040] := 16#763F;
   // UNICODE_TO_GBK[22041] := 16#F1A8;
   // UNICODE_TO_GBK[22042] := 16#7640;
   // UNICODE_TO_GBK[22043] := 16#F1A5;
   // UNICODE_TO_GBK[22044] := 16#7641;
   // UNICODE_TO_GBK[22045] := 16#AF9E;
   // UNICODE_TO_GBK[22046] := 16#7642;
   // UNICODE_TO_GBK[22047] := 16#AF9F;
   // UNICODE_TO_GBK[22048] := 16#7643;
   // UNICODE_TO_GBK[22049] := 16#F1AA;
   // UNICODE_TO_GBK[22050] := 16#7644;
   // UNICODE_TO_GBK[22051] := 16#AFA0;
   // UNICODE_TO_GBK[22052] := 16#7645;
   // UNICODE_TO_GBK[22053] := 16#B040;
   // UNICODE_TO_GBK[22054] := 16#7646;
   // UNICODE_TO_GBK[22055] := 16#B041;
   // UNICODE_TO_GBK[22056] := 16#7647;
   // UNICODE_TO_GBK[22057] := 16#B042;
   // UNICODE_TO_GBK[22058] := 16#7648;
   // UNICODE_TO_GBK[22059] := 16#B043;
   // UNICODE_TO_GBK[22060] := 16#7649;
   // UNICODE_TO_GBK[22061] := 16#B044;
   // UNICODE_TO_GBK[22062] := 16#764A;
   // UNICODE_TO_GBK[22063] := 16#B045;
   // UNICODE_TO_GBK[22064] := 16#764B;
   // UNICODE_TO_GBK[22065] := 16#B046;
   // UNICODE_TO_GBK[22066] := 16#764C;
   // UNICODE_TO_GBK[22067] := 16#B0A9;
   // UNICODE_TO_GBK[22068] := 16#764D;
   // UNICODE_TO_GBK[22069] := 16#F1AD;
   // UNICODE_TO_GBK[22070] := 16#764E;
   // UNICODE_TO_GBK[22071] := 16#B047;
   // UNICODE_TO_GBK[22072] := 16#764F;
   // UNICODE_TO_GBK[22073] := 16#B048;
   // UNICODE_TO_GBK[22074] := 16#7650;
   // UNICODE_TO_GBK[22075] := 16#B049;
   // UNICODE_TO_GBK[22076] := 16#7651;
   // UNICODE_TO_GBK[22077] := 16#B04A;
   // UNICODE_TO_GBK[22078] := 16#7652;
   // UNICODE_TO_GBK[22079] := 16#B04B;
   // UNICODE_TO_GBK[22080] := 16#7653;
   // UNICODE_TO_GBK[22081] := 16#B04C;
   // UNICODE_TO_GBK[22082] := 16#7654;
   // UNICODE_TO_GBK[22083] := 16#F1AF;
   // UNICODE_TO_GBK[22084] := 16#7655;
   // UNICODE_TO_GBK[22085] := 16#B04D;
   // UNICODE_TO_GBK[22086] := 16#7656;
   // UNICODE_TO_GBK[22087] := 16#F1B1;
   // UNICODE_TO_GBK[22088] := 16#7657;
   // UNICODE_TO_GBK[22089] := 16#B04E;
   // UNICODE_TO_GBK[22090] := 16#7658;
   // UNICODE_TO_GBK[22091] := 16#B04F;
   // UNICODE_TO_GBK[22092] := 16#7659;
   // UNICODE_TO_GBK[22093] := 16#B050;
   // UNICODE_TO_GBK[22094] := 16#765A;
   // UNICODE_TO_GBK[22095] := 16#B051;
   // UNICODE_TO_GBK[22096] := 16#765B;
   // UNICODE_TO_GBK[22097] := 16#B052;
   // UNICODE_TO_GBK[22098] := 16#765C;
   // UNICODE_TO_GBK[22099] := 16#F1B0;
   // UNICODE_TO_GBK[22100] := 16#765D;
   // UNICODE_TO_GBK[22101] := 16#B053;
   // UNICODE_TO_GBK[22102] := 16#765E;
   // UNICODE_TO_GBK[22103] := 16#F1AE;
   // UNICODE_TO_GBK[22104] := 16#765F;
   // UNICODE_TO_GBK[22105] := 16#B054;
   // UNICODE_TO_GBK[22106] := 16#7660;
   // UNICODE_TO_GBK[22107] := 16#B055;
   // UNICODE_TO_GBK[22108] := 16#7661;
   // UNICODE_TO_GBK[22109] := 16#B056;
   // UNICODE_TO_GBK[22110] := 16#7662;
   // UNICODE_TO_GBK[22111] := 16#B057;
   // UNICODE_TO_GBK[22112] := 16#7663;
   // UNICODE_TO_GBK[22113] := 16#D1A2;
   // UNICODE_TO_GBK[22114] := 16#7664;
   // UNICODE_TO_GBK[22115] := 16#B058;
   // UNICODE_TO_GBK[22116] := 16#7665;
   // UNICODE_TO_GBK[22117] := 16#B059;
   // UNICODE_TO_GBK[22118] := 16#7666;
   // UNICODE_TO_GBK[22119] := 16#B05A;
   // UNICODE_TO_GBK[22120] := 16#7667;
   // UNICODE_TO_GBK[22121] := 16#B05B;
   // UNICODE_TO_GBK[22122] := 16#7668;
   // UNICODE_TO_GBK[22123] := 16#B05C;
   // UNICODE_TO_GBK[22124] := 16#7669;
   // UNICODE_TO_GBK[22125] := 16#B05D;
   // UNICODE_TO_GBK[22126] := 16#766A;
   // UNICODE_TO_GBK[22127] := 16#B05E;
   // UNICODE_TO_GBK[22128] := 16#766B;
   // UNICODE_TO_GBK[22129] := 16#F1B2;
   // UNICODE_TO_GBK[22130] := 16#766C;
   // UNICODE_TO_GBK[22131] := 16#B05F;
   // UNICODE_TO_GBK[22132] := 16#766D;
   // UNICODE_TO_GBK[22133] := 16#B060;
   // UNICODE_TO_GBK[22134] := 16#766E;
   // UNICODE_TO_GBK[22135] := 16#B061;
   // UNICODE_TO_GBK[22136] := 16#766F;
   // UNICODE_TO_GBK[22137] := 16#F1B3;
   // UNICODE_TO_GBK[22138] := 16#7670;
   // UNICODE_TO_GBK[22139] := 16#B062;
   // UNICODE_TO_GBK[22140] := 16#7671;
   // UNICODE_TO_GBK[22141] := 16#B063;
   // UNICODE_TO_GBK[22142] := 16#7672;
   // UNICODE_TO_GBK[22143] := 16#B064;
   // UNICODE_TO_GBK[22144] := 16#7673;
   // UNICODE_TO_GBK[22145] := 16#B065;
   // UNICODE_TO_GBK[22146] := 16#7674;
   // UNICODE_TO_GBK[22147] := 16#B066;
   // UNICODE_TO_GBK[22148] := 16#7675;
   // UNICODE_TO_GBK[22149] := 16#B067;
   // UNICODE_TO_GBK[22150] := 16#7676;
   // UNICODE_TO_GBK[22151] := 16#B068;
   // UNICODE_TO_GBK[22152] := 16#7677;
   // UNICODE_TO_GBK[22153] := 16#B069;
   // UNICODE_TO_GBK[22154] := 16#7678;
   // UNICODE_TO_GBK[22155] := 16#B9EF;
   // UNICODE_TO_GBK[22156] := 16#7679;
   // UNICODE_TO_GBK[22157] := 16#B06A;
   // UNICODE_TO_GBK[22158] := 16#767A;
   // UNICODE_TO_GBK[22159] := 16#B06B;
   // UNICODE_TO_GBK[22160] := 16#767B;
   // UNICODE_TO_GBK[22161] := 16#B5C7;
   // UNICODE_TO_GBK[22162] := 16#767C;
   // UNICODE_TO_GBK[22163] := 16#B06C;
   // UNICODE_TO_GBK[22164] := 16#767D;
   // UNICODE_TO_GBK[22165] := 16#B0D7;
   // UNICODE_TO_GBK[22166] := 16#767E;
   // UNICODE_TO_GBK[22167] := 16#B0D9;
   // UNICODE_TO_GBK[22168] := 16#767F;
   // UNICODE_TO_GBK[22169] := 16#B06D;
   // UNICODE_TO_GBK[22170] := 16#7680;
   // UNICODE_TO_GBK[22171] := 16#B06E;
   // UNICODE_TO_GBK[22172] := 16#7681;
   // UNICODE_TO_GBK[22173] := 16#B06F;
   // UNICODE_TO_GBK[22174] := 16#7682;
   // UNICODE_TO_GBK[22175] := 16#D4ED;
   // UNICODE_TO_GBK[22176] := 16#7683;
   // UNICODE_TO_GBK[22177] := 16#B070;
   // UNICODE_TO_GBK[22178] := 16#7684;
   // UNICODE_TO_GBK[22179] := 16#B5C4;
   // UNICODE_TO_GBK[22180] := 16#7685;
   // UNICODE_TO_GBK[22181] := 16#B071;
   // UNICODE_TO_GBK[22182] := 16#7686;
   // UNICODE_TO_GBK[22183] := 16#BDD4;
   // UNICODE_TO_GBK[22184] := 16#7687;
   // UNICODE_TO_GBK[22185] := 16#BBCA;
   // UNICODE_TO_GBK[22186] := 16#7688;
   // UNICODE_TO_GBK[22187] := 16#F0A7;
   // UNICODE_TO_GBK[22188] := 16#7689;
   // UNICODE_TO_GBK[22189] := 16#B072;
   // UNICODE_TO_GBK[22190] := 16#768A;
   // UNICODE_TO_GBK[22191] := 16#B073;
   // UNICODE_TO_GBK[22192] := 16#768B;
   // UNICODE_TO_GBK[22193] := 16#B8DE;
   // UNICODE_TO_GBK[22194] := 16#768C;
   // UNICODE_TO_GBK[22195] := 16#B074;
   // UNICODE_TO_GBK[22196] := 16#768D;
   // UNICODE_TO_GBK[22197] := 16#B075;
   // UNICODE_TO_GBK[22198] := 16#768E;
   // UNICODE_TO_GBK[22199] := 16#F0A8;
   // UNICODE_TO_GBK[22200] := 16#768F;
   // UNICODE_TO_GBK[22201] := 16#B076;
   // UNICODE_TO_GBK[22202] := 16#7690;
   // UNICODE_TO_GBK[22203] := 16#B077;
   // UNICODE_TO_GBK[22204] := 16#7691;
   // UNICODE_TO_GBK[22205] := 16#B0A8;
   // UNICODE_TO_GBK[22206] := 16#7692;
   // UNICODE_TO_GBK[22207] := 16#B078;
   // UNICODE_TO_GBK[22208] := 16#7693;
   // UNICODE_TO_GBK[22209] := 16#F0A9;
   // UNICODE_TO_GBK[22210] := 16#7694;
   // UNICODE_TO_GBK[22211] := 16#B079;
   // UNICODE_TO_GBK[22212] := 16#7695;
   // UNICODE_TO_GBK[22213] := 16#B07A;
   // UNICODE_TO_GBK[22214] := 16#7696;
   // UNICODE_TO_GBK[22215] := 16#CDEE;
   // UNICODE_TO_GBK[22216] := 16#7697;
   // UNICODE_TO_GBK[22217] := 16#B07B;
   // UNICODE_TO_GBK[22218] := 16#7698;
   // UNICODE_TO_GBK[22219] := 16#B07C;
   // UNICODE_TO_GBK[22220] := 16#7699;
   // UNICODE_TO_GBK[22221] := 16#F0AA;
   // UNICODE_TO_GBK[22222] := 16#769A;
   // UNICODE_TO_GBK[22223] := 16#B07D;
   // UNICODE_TO_GBK[22224] := 16#769B;
   // UNICODE_TO_GBK[22225] := 16#B07E;
   // UNICODE_TO_GBK[22226] := 16#769C;
   // UNICODE_TO_GBK[22227] := 16#B080;
   // UNICODE_TO_GBK[22228] := 16#769D;
   // UNICODE_TO_GBK[22229] := 16#B081;
   // UNICODE_TO_GBK[22230] := 16#769E;
   // UNICODE_TO_GBK[22231] := 16#B082;
   // UNICODE_TO_GBK[22232] := 16#769F;
   // UNICODE_TO_GBK[22233] := 16#B083;
   // UNICODE_TO_GBK[22234] := 16#76A0;
   // UNICODE_TO_GBK[22235] := 16#B084;
   // UNICODE_TO_GBK[22236] := 16#76A1;
   // UNICODE_TO_GBK[22237] := 16#B085;
   // UNICODE_TO_GBK[22238] := 16#76A2;
   // UNICODE_TO_GBK[22239] := 16#B086;
   // UNICODE_TO_GBK[22240] := 16#76A3;
   // UNICODE_TO_GBK[22241] := 16#B087;
   // UNICODE_TO_GBK[22242] := 16#76A4;
   // UNICODE_TO_GBK[22243] := 16#F0AB;
   // UNICODE_TO_GBK[22244] := 16#76A5;
   // UNICODE_TO_GBK[22245] := 16#B088;
   // UNICODE_TO_GBK[22246] := 16#76A6;
   // UNICODE_TO_GBK[22247] := 16#B089;
   // UNICODE_TO_GBK[22248] := 16#76A7;
   // UNICODE_TO_GBK[22249] := 16#B08A;
   // UNICODE_TO_GBK[22250] := 16#76A8;
   // UNICODE_TO_GBK[22251] := 16#B08B;
   // UNICODE_TO_GBK[22252] := 16#76A9;
   // UNICODE_TO_GBK[22253] := 16#B08C;
   // UNICODE_TO_GBK[22254] := 16#76AA;
   // UNICODE_TO_GBK[22255] := 16#B08D;
   // UNICODE_TO_GBK[22256] := 16#76AB;
   // UNICODE_TO_GBK[22257] := 16#B08E;
   // UNICODE_TO_GBK[22258] := 16#76AC;
   // UNICODE_TO_GBK[22259] := 16#B08F;
   // UNICODE_TO_GBK[22260] := 16#76AD;
   // UNICODE_TO_GBK[22261] := 16#B090;
   // UNICODE_TO_GBK[22262] := 16#76AE;
   // UNICODE_TO_GBK[22263] := 16#C6A4;
   // UNICODE_TO_GBK[22264] := 16#76AF;
   // UNICODE_TO_GBK[22265] := 16#B091;
   // UNICODE_TO_GBK[22266] := 16#76B0;
   // UNICODE_TO_GBK[22267] := 16#B092;
   // UNICODE_TO_GBK[22268] := 16#76B1;
   // UNICODE_TO_GBK[22269] := 16#D6E5;
   // UNICODE_TO_GBK[22270] := 16#76B2;
   // UNICODE_TO_GBK[22271] := 16#F1E4;
   // UNICODE_TO_GBK[22272] := 16#76B3;
   // UNICODE_TO_GBK[22273] := 16#B093;
   // UNICODE_TO_GBK[22274] := 16#76B4;
   // UNICODE_TO_GBK[22275] := 16#F1E5;
   // UNICODE_TO_GBK[22276] := 16#76B5;
   // UNICODE_TO_GBK[22277] := 16#B094;
   // UNICODE_TO_GBK[22278] := 16#76B6;
   // UNICODE_TO_GBK[22279] := 16#B095;
   // UNICODE_TO_GBK[22280] := 16#76B7;
   // UNICODE_TO_GBK[22281] := 16#B096;
   // UNICODE_TO_GBK[22282] := 16#76B8;
   // UNICODE_TO_GBK[22283] := 16#B097;
   // UNICODE_TO_GBK[22284] := 16#76B9;
   // UNICODE_TO_GBK[22285] := 16#B098;
   // UNICODE_TO_GBK[22286] := 16#76BA;
   // UNICODE_TO_GBK[22287] := 16#B099;
   // UNICODE_TO_GBK[22288] := 16#76BB;
   // UNICODE_TO_GBK[22289] := 16#B09A;
   // UNICODE_TO_GBK[22290] := 16#76BC;
   // UNICODE_TO_GBK[22291] := 16#B09B;
   // UNICODE_TO_GBK[22292] := 16#76BD;
   // UNICODE_TO_GBK[22293] := 16#B09C;
   // UNICODE_TO_GBK[22294] := 16#76BE;
   // UNICODE_TO_GBK[22295] := 16#B09D;
   // UNICODE_TO_GBK[22296] := 16#76BF;
   // UNICODE_TO_GBK[22297] := 16#C3F3;
   // UNICODE_TO_GBK[22298] := 16#76C0;
   // UNICODE_TO_GBK[22299] := 16#B09E;
   // UNICODE_TO_GBK[22300] := 16#76C1;
   // UNICODE_TO_GBK[22301] := 16#B09F;
   // UNICODE_TO_GBK[22302] := 16#76C2;
   // UNICODE_TO_GBK[22303] := 16#D3DB;
   // UNICODE_TO_GBK[22304] := 16#76C3;
   // UNICODE_TO_GBK[22305] := 16#B0A0;
   // UNICODE_TO_GBK[22306] := 16#76C4;
   // UNICODE_TO_GBK[22307] := 16#B140;
   // UNICODE_TO_GBK[22308] := 16#76C5;
   // UNICODE_TO_GBK[22309] := 16#D6D1;
   // UNICODE_TO_GBK[22310] := 16#76C6;
   // UNICODE_TO_GBK[22311] := 16#C5E8;
   // UNICODE_TO_GBK[22312] := 16#76C7;
   // UNICODE_TO_GBK[22313] := 16#B141;
   // UNICODE_TO_GBK[22314] := 16#76C8;
   // UNICODE_TO_GBK[22315] := 16#D3AF;
   // UNICODE_TO_GBK[22316] := 16#76C9;
   // UNICODE_TO_GBK[22317] := 16#B142;
   // UNICODE_TO_GBK[22318] := 16#76CA;
   // UNICODE_TO_GBK[22319] := 16#D2E6;
   // UNICODE_TO_GBK[22320] := 16#76CB;
   // UNICODE_TO_GBK[22321] := 16#B143;
   // UNICODE_TO_GBK[22322] := 16#76CC;
   // UNICODE_TO_GBK[22323] := 16#B144;
   // UNICODE_TO_GBK[22324] := 16#76CD;
   // UNICODE_TO_GBK[22325] := 16#EEC1;
